"IX_ROBOT_PROT_DOOR_CLSD"	I 3111.3	BOOL	// F4-66.7 Werkstücklader Schutzzaun geschlossen
"MSST_Vorschub_OVR"	IB 3	BYTE	// Maschinensteuertafel Vorschub Override
"MSST_Eilgang_OVR"	IB 7	BYTE	// Maschinensteuertafel Eilgang Override
"IX_Direkttasten_links"	IB 8	BYTE	// HMI-PRO: OP12/OP15A Direkttasten links
"IX_Direkttasten_rechts"	IB 9	BYTE	// HMI-PRO: OP12/OP15A Direkttasten rechts
"IW_SPI_VIBRATION"	IW 100	WORD	// Analogeingang Vibrationssensor
"IW_FD_PT100"	IW 156	WORD	// Temperatursensor Pt100 Fraes-Drehtisch
"IW_MI_TURNT_TEMP"	IW 1000	WORD	// Temp.-Sensor PT100 Fraes-Drehtisch
"IW_MACH_BED_T_COMP"	IW 1090	WORD
"IW_SPI_TEMP_BEA_FRONT"	IW 1092	WORD
"IW_VMS_VIBRATION_SPINDLE"	IW 1094	WORD
"IW_SPI_LINE_PT100_1"	IW 1102	WORD	// Temperatursensor 1 Leitungsueberwachung Hauptantrieb
"IW_SPI_LINE_PT100_2"	IW 1104	WORD	// Temperatursensor 2 Leitungsueberwachung Hauptantrieb
"IW_SPI_PT100"	IW 1106	WORD	// Lager-Temperatursensor PT100 Hauptantrieb
"IW_HCD_PRE_MPL"	IW 1108	WORD	// Spannhydraulik Druckueberwachung Maschine
"IW_HCD_PRE_SST"	IW 1110	WORD	// Spannhydraulik Druckueberwachung Ruestplatz
"IW_SPI_TEMP_LAG_VORNE"	IW 1112	WORD	// Lager-Temperatursensor PT100 Hauptantrieb
"IW_SPI_TEMP_LAG_HINTEN"	IW 1122	WORD	// Lager-Temperatursensor PT100 Hauptantrieb
"IW_SPI_TEMP_MONITOR"	IW 2000	WORD	// Temperaturüberwachung Spindelstock (55/65H)
"IW_RESERVE_4_33"	IW 2002	WORD	// Dummy für Hardware 55H
"BT_ET200S_3_12"	IW 3106	WORD	// E5-03.5 Analogeingang Reserve
"BT_ET200S_4_5"	IW 3108	WORD	// Analogeingang Reserve
"m_null"	M 0.0	BOOL	// Status 0
"m_eins"	M 0.1	BOOL	// Status 1
"m_expertenbit"	M 0.2	BOOL	// Expertenbit für Fehleranzeige
"m_dummy"	M 0.3	BOOL	// Dummy
"m_vke_uebertrag_1"	M 0.4	BOOL	// VKE Übertrag 1
"m_neustart"	M 0.5	BOOL	// Neustart
"m_inbetrieb_logisch_1"	M 0.6	BOOL	// Inbetriebnahmemerker Logisch 1
"m_konstruktion"	M 0.7	BOOL	// Konstruktionsmerker Logisch 1
"m_takt_0,1sec."	M 1.0	BOOL	// Taktmerker System 100 ms
"m_takt_0,2sec."	M 1.1	BOOL	// Taktmerker System 200 ms
"m_takt_0,4sec."	M 1.2	BOOL	// Taktmerker System 400 ms
"m_takt_0,5sec."	M 1.3	BOOL	// Taktmerker System 500 ms
"m_takt_0,8sec."	M 1.4	BOOL	// Taktmerker System 800 ms
"m_takt_1sec."	M 1.5	BOOL	// Taktmerker System 1000 ms
"m_takt_1,6sec."	M 1.6	BOOL	// Taktmerker System 1600 ms
"m_takt_2sec."	M 1.7	BOOL	// Taktmerker System 2000 ms
"M_1_ter_OB1_Zyklus"	M 2.0	BOOL	// Erster Zyklus OrganisationsBaustein 1
"M_2_ter_OB1_Zyklus"	M 2.1	BOOL	// Zweiter Zyklus OrganisationsBaustein 1
"M_3_ter_OB1_Zyklus"	M 2.2	BOOL	// Dritter Zyklus OrganisationsBaustein 1
"M_4_ter_OB1_Zyklus"	M 2.3	BOOL	// Vierter Zyklus OrganisationsBaustein 1
"M_5_ter_OB1_Zyklus"	M 2.4	BOOL	// Fünfter Zyklus OrganisationsBaustein 1
"M_6_ter_OB1_Zyklus"	M 2.5	BOOL	// Sechster Zyklus OrganisationsBaustein 1
"M_7_ter_OB1_Zyklus"	M 2.6	BOOL	// Siebter Zyklus OrganisationsBaustein 1
"M_8_ter_OB1_Zyklen"	M 2.7	BOOL	// Achter Zyklus OrganisationsBaustein 1
"M_CHAN2_aktiv"	M 6.0	BOOL	// Kanal 2 aktiv
"m_6.1"	M 6.1	BOOL	// Reserve
"m_6.2"	M 6.2	BOOL	// Reserve
"m_6.3"	M 6.3	BOOL	// Reserve
"m_6.4"	M 6.4	BOOL	// Reserve
"m_6.5"	M 6.5	BOOL	// Reserve
"m_6.6"	M 6.6	BOOL	// Reserve
"M_Takt_10s"	M 6.7	BOOL	// Taktmerker 10 s
"M_Takt_01s"	M 7.0	BOOL	// Taktmerker 100 ms
"M_Takt_02s"	M 7.1	BOOL	// Taktmerker 200 ms
"M_Takt_04s"	M 7.2	BOOL	// Taktmerker 400 ms
"M_Takt_05s"	M 7.3	BOOL	// Taktmerker 500 ms
"M_Takt_08s"	M 7.4	BOOL	// Taktmerker 800 ms
"M_Takt_1s"	M 7.5	BOOL	// Taktmerker 1000 ms
"M_Takt_16s"	M 7.6	BOOL	// Taktmerker 1600 ms
"M_Takt_2s"	M 7.7	BOOL	// Taktmerker 2000 ms
"M_Takt_Speicher_01s"	M 8.0	BOOL	// Taktmerker Speicher 100 ms
"M_Takt_Speicher_02s"	M 8.1	BOOL	// Taktmerker Speicher 200 ms
"M_Takt_Speicher_04s"	M 8.2	BOOL	// Taktmerker Speicher 400 ms
"M_Takt_Speicher_05s"	M 8.3	BOOL	// Taktmerker Speicher 500 ms
"M_Takt_Speicher_08s"	M 8.4	BOOL	// Taktmerker Speicher 800 ms
"M_Takt_Speicher_1s"	M 8.5	BOOL	// TaktmerkerSpeicher 1000 ms
"M_Takt_Speicher_16s"	M 8.6	BOOL	// Taktmerker Speicher 1600 ms
"M_Takt_Speicher_2s"	M 8.7	BOOL	// Taktmerker Speicher 2000 ms
"M_1_ter_OB1_Zyklus_stat"	M 9.0	BOOL	// Erster Zyklus OrganisationsBaustein 1
"M_Ruecksetze_Fehler"	M 10.0	BOOL	// Globaler Reset fuer Fehler (Quitt Taste und Reset Taste)
"M_NC_Stop"	M 10.1	BOOL	// Globaler NC Stop
"M_Vorschub_Halt_Kanal"	M 10.2	BOOL	// Globaler Vorschub Halt
"M_Spindel_Halt_Kanal"	M 10.3	BOOL	// Globaler Spindel Halt
"M_Vorschub_Halt_Haupt"	M 10.4	BOOL	// Vorschub Halt Hauptachsen
"M_Reset_Taste"	M 10.5	BOOL	// Globaler Impuls Reset Taste
"M_Fehler_Quit_Taste"	M 10.6	BOOL	// Globaler Impuls Quittier Taste
"M_NC_Stop_Taste"	M 10.7	BOOL	// NC-Stop Taste in BA AUTO (nicht in Jog)
"M_NC_Start_Taste"	M 11.0	BOOL	// NC-Start Taste in BA AUTO (nicht in Jog)
"M_Spindel_Sperre_Auto"	M 11.1	BOOL	// Spindel-Sperre Taste in Automatik
"M_Vorschub_Sperre_Auto"	M 11.2	BOOL	// Vorschub-Sperre Taste in Automatik
"M_Eilgang_verriegeln"	M 11.3	BOOL	// Eilgangtaste verriegeln
"M_Vorschub_Halt_Asyn1"	M 11.4	BOOL	// Vorschub Halt Asynchroner Prozess 1 (701548-701631 -> Mag: Achse 7)
"M_Vorschub_Halt_Asyn2"	M 11.5	BOOL	// Vorschub Halt Asynchroner Prozess 2 (701632-701715 -> PW: Achse 8)
"M_Vorschub_Halt_Asyn3"	M 11.6	BOOL	// Vorschub Halt Asynchroner Prozess 3 (701716-701763 -> Pal.Speicher: Achse9/10)
"M_Vorschub_Halt_Asyn4"	M 11.7	BOOL	// Vorschub Halt Asynchroner Prozess 4 (701800-701847 ->  Mag: Achse 7)
"M_Handbetrieb"	M 12.0	BOOL	// Manual / Jog-betrieb steht an
"M_Satzfolge_aktiv"	M 12.1	BOOL	// Automatikbetrieb
"M_Einzelsatz"	M 12.2	BOOL	// Einzelsatz
"M_Simulation_Aktiv"	M 12.3	BOOL	// Simulation Aktiv
"M_Programm_Aktiv"	M 12.4	BOOL	// Programm Aktiv
"M_Hauptprogramm_Ende"	M 12.5	BOOL	// Hauptprogramm Ende
"M_HM_Hauptprogramm_Ende"	M 12.6	BOOL	// Hilfsmerker Hauptprogramm Ende
"M_Gewindeschneiden_aktiv"	M 12.7	BOOL	// Nahtstelle: Gewindeschneiden aktiv
"M_Hauptspindel_steht"	M 13.0	BOOL	// Hauptspindel steht
"M_Hauptachsen_stehen"	M 13.1	BOOL	// Hauptachsen stehen
"M_ShopMill_aktiv"	M 13.2	BOOL	// ShopMill Bedienoberflaeche aktiv
"M_FahrAnf_HauptAchs"	M 13.3	BOOL	// Fahranforderung Hauptachsen steht an
"M_G00_aktiv"	M 13.4	BOOL	// G0 Aktiv
"M_G02_G03_aktiv"	M 13.5	BOOL	// G02 oder G03 Aktiv
"M_G74_aktiv"	M 13.6	BOOL	// G74 Aktiv
"M_Automatik_Betrieb"	M 13.7	BOOL	// Automatikbetrieb steht an
"M_ShopMill_Manual"	M 14.0	BOOL	// ShopMill im Manual
"M_ShopMill_Positionieren"	M 14.1	BOOL	// ShopMill Positionieren
"MX_MsSt_Vorschub_0"	M 14.2	BOOL	// Anforderung MSST Vorschub Override auf 0
"MX_M0_1_Aktiv"	M 14.3	BOOL	// M0 oder M1 ist aktiv
"MX_Flanke_M01"	M 14.4	BOOL	// Flanke Positiv M0 M1
"MX_MDA"	M 14.5	BOOL	// MDA Aktiv
"MX_FN_Leistung_Steht_an"	M 14.6	BOOL	// Flanke Negativ Leistung
"MX_IMP_Leistung_0"	M 14.7	BOOL	// Flanke Negativ Leistung Steht an
"MX_SonderBA_Stop"	M 15.0	BOOL	// Stop Aktiv nach verlassen der Sonder BA's
"MX_PLC_Initialisiert"	M 15.1	BOOL	// PLC Initialisiert
"M_Programm_Aktiv_Kanal_1"	M 15.2	BOOL	// Programm aktiv im Kanal 1(Run/Wait/Stop/Interrupt)
"MX_Satzsuchlauf_gesp"	M 15.3	BOOL	// Satzsuchlauf aktiv gespeichert
"O_PW_TUER_ENTRIEGELN"	M 15.4	BOOL	// M-AUSGANG: Magnetverriegelung Ruestplatz Palettenwechsler verriegeln
"O_PW_Ventil_Abfrage"	M 15.5	BOOL	// M-AUSGANG: Ventil Luftstrom Palette
"M_G01_aktiv"	M 15.6	BOOL	// G1 Aktiv
"O_PW_Ventil_Tischspuel"	M 15.7	BOOL	// M-AUSGANG: IKZ-Pumpe ein für Tischspuelung
"I_MSST_PW_Freigabe"	M 16.0	BOOL	// M-EINGANG: Eingang Freigabe Palettenwechsler
"I_PW_MPL_belegt"	M 16.1	BOOL	// M-EINGANG: Palette in der Maschine vorhanden
"I_PW_Ruestpl_UeberG"	M 16.2	BOOL	// M-EINGANG: Palette Übergabeplatz Maschine
"I_PW_Hub_in_Mitte"	M 16.3	BOOL	// M-EINGANG: Palettenwechsler Hub Pos. Mitte
"I_PW_Tueren_verriegelt"	M 16.4	BOOL	// M-EINGANG: Fenster Ruestplatz PW verriegelt
"I_PW_Klemmung_Geklemmt"	M 16.5	BOOL	// M-EINGANG: Palettenklemmung geklemmt
"I_PW_Klemmung_Gelöst"	M 16.6	BOOL	// M-EINGANG: Palettenklemmung gelöst
"M_FLANKE_START_TASTE"	M 16.7	BOOL	// Flanke Positiv NC-Start Taste
"M_Flanke_M208"	M 17.0	BOOL	// TEMPERATURKOMPENSATION: M-Funktion 208 Flanke positiv
"M_Flanke_M209"	M 17.1	BOOL	// TEMPERATURKOMPENSATION: M-Funktion 209 Flanke positiv
"M_Umlaufzaehler=0"	M 17.3	BOOL	// TEMPERATURKOMPENSATION: Umlaufzähler HM
"M_Zyklus_Takt"	M 17.4	BOOL	// TEMPERATURKOMPENSATION: Zyklus Takt
"M_VSH_ASYN_DISABLE_START"	M 17.5	BOOL	// Ersten Start unterdrücken nach Vorschub Halt Asynchroner Prozess bei Fertigtteil
"m_17.6"	M 17.6	BOOL	// Reserve
"M_Fuehlerumschaltung"	M 17.7	BOOL	// TEMPERATURKOMPENSATION: Fühlerumschaltung
"M_Trend_Temp_auf"	M 18.0	BOOL	// TEMPERATURKOMPENSATION: Temperaturtrend aufwärts
"M_Trend_Temp_gleich"	M 18.1	BOOL	// TEMPERATURKOMPENSATION: Temperaturtrend gleichbleibend
"M_Trend_Temp_ab"	M 18.2	BOOL	// TEMPERATURKOMPENSATION: Temperaturtrend abwärts
"M_Fehler_Temp-Tabelle"	M 18.3	BOOL	// TEMPERATURKOMPENSATION: Fehler Temperaturtabelle
"M_FM_Timer_Verzoegerung"	M 18.4	BOOL	// TEMPERATURKOMPENSATION: Timer Verzögerung
"M_FP_Timer_Verzoegerung"	M 18.5	BOOL	// TEMPERATURKOMPENSATION: Timer Verzögerung Flanke positiv
"M_Temp-Daten_uebertragen"	M 18.6	BOOL	// TEMPERATURKOMPENSATION: Temperaturdaten übertragen
"M_MesswertInterv_0"	M 18.7	BOOL	// TEMPERATURKOMPENSATION: Messwert-Intervall  = 0
"M_Trend_Drehz_auf"	M 19.0	BOOL	// TEMPERATURKOMPENSATION: Drehzahltrend aufwärts
"M_Trend_Drehz_gleich"	M 19.1	BOOL	// TEMPERATURKOMPENSATION: Drehzahltrend gleichbleibend
"M_Trend_Drehz_ab"	M 19.2	BOOL	// TEMPERATURKOMPENSATION: Drehzahltrend abwärts
"M_Fehler_Drehz-Tabelle"	M 19.3	BOOL	// TEMPERATURKOMPENSATION: Fehler Drehzahltabelle
"M_Temp_Wert <"	M 19.4	BOOL	// TEMPERATURKOMPENSATION: Temperaturwert kleiner
"M_Temp_Wert ="	M 19.5	BOOL	// TEMPERATURKOMPENSATION: Temperaturwert gleich
"M_Temp_Wert >"	M 19.6	BOOL	// TEMPERATURKOMPENSATION: Temperaturwert größer
"HM_PI_Umlauf"	M 19.7	BOOL	// TEMPERATURKOMPENSATION:  PI Umlaufzähler = 0 Flanke positiv
"M_FP_Einrichtb"	M 20.0	BOOL	// Einrichtbetrieb Flanke positiv
"M_Imp_Einrichtberieb"	M 20.1	BOOL	// Einrichtbetrieb Impuls
"M_FP_BA3"	M 20.2	BOOL	// Betriebsart 3 Flanke positiv
"M_Imp_Betriebsart 3"	M 20.3	BOOL	// Betriebsart 3  Impuls
"M_FP_BA4+ZUSTT"	M 20.4	BOOL	// Betriebsart 4 Flanke positiv
"M_BA4_aktiv_schalten_"	M 20.5	BOOL	// Betriebsart 4  aktiv
"m_20.6"	M 20.6	BOOL	// Reserve
"m_20.7"	M 20.7	BOOL	// Reserve
"m_21.0"	M 21.0	BOOL	// Reserve
"m_21.1"	M 21.1	BOOL	// Reserve
"m_21.2"	M 21.2	BOOL	// Reserve
"m_21.3"	M 21.3	BOOL	// Reserve
"m_21.4"	M 21.4	BOOL	// Reserve
"m_21.5"	M 21.5	BOOL	// Reserve
"m_21.6"	M 21.6	BOOL	// Reserve
"m_21.7"	M 21.7	BOOL	// Reserve
"m_22.0"	M 22.0	BOOL	// Reserve
"M_Selbsth_AT_X-plus"	M 22.1	BOOL	// MSTT: Selbsthaltung für Achsenkreuztaste X-Plus
"M_Selbsth_AT_X-minus"	M 22.2	BOOL	// MSTT: Selbsthaltung für Achsenkreuztaste X-Minus
"m_22.3"	M 22.3	BOOL	// Reserve
"m_22.4"	M 22.4	BOOL	// Reserve
"m_22.5"	M 22.5	BOOL	// Reserve
"m_22.6"	M 22.6	BOOL	// Reserve
"m_22.7"	M 22.7	BOOL	// Reserve
"m_23.0"	M 23.0	BOOL	// Reserve
"m_23.1"	M 23.1	BOOL	// Reserve
"M_Selbsth_AT_Y-minus"	M 23.2	BOOL	// MSTT: Selbsthaltung für Achsenkreuztaste Y-Minus
"M_Selbsth_AT_Y-plus"	M 23.3	BOOL	// MSTT: Selbsthaltung für Achsenkreuztaste Y-Plus
"M_Selbsth_AT_Z-minus"	M 23.4	BOOL	// MSTT: Selbsthaltung für Achsenkreuztaste Z-Minus
"M_Selbsth_AT_Z-plus"	M 23.5	BOOL	// MSTT: Selbsthaltung für Achsenkreuztaste Z-Plus
"M_Selbsth_AT_4-minus"	M 23.6	BOOL	// MSTT: Selbsthaltung für Achsenkreuztaste 4-Minus
"M_Selbsth_AT_4-plus"	M 23.7	BOOL	// MSTT: Selbsthaltung für Achsenkreuztaste 4-Plus
"M_Selbsth_AT_5-minus"	M 24.0	BOOL	// MSTT: Selbsthaltung für Achsenkreuztaste 5-Minus
"M_Selbsth_AT_5-plus"	M 24.1	BOOL	// MSTT: Selbsthaltung für Achsenkreuztaste 5-Plus
"M_Selbsth_AT_6-minus"	M 24.2	BOOL	// MSTT: Selbsthaltung für Achsenkreuztaste 6-Minus
"M_Selbsth_AT_6-plus"	M 24.3	BOOL	// MSTT: Selbsthaltung für Achsenkreuztaste 6-Plus
"M_Selbsth_AT_10-minus"	M 24.4	BOOL	// MSTT: Selbsthaltung für Achsenkreuztaste 10-Minus
"M_Selbsth_AT_10-plus"	M 24.5	BOOL	// MSTT: Selbsthaltung für Achsenkreuztaste 10-Plus
"O_SP_RPL_MPL_BLASLUFT"	M 24.6	BOOL	// M-AUSGANG: Ventil Blasluft Medienkupplung
"M_FP_mxplus"	M 24.7	BOOL	// Flanke Positiv Achsenkreuztaste X-Plus
"M_FP_mxminus"	M 25.0	BOOL	// Flanke Positiv Achsenkreuztaste X-Minus
"M_FP_myplus"	M 25.1	BOOL	// Flanke Positiv Achsenkreuztaste Y-Plus
"M_FP_myminus"	M 25.2	BOOL	// Flanke Positiv Achsenkreuztaste Y-Minus
"M_FP_mzplus"	M 25.3	BOOL	// Flanke Positiv Achsenkreuztaste Z-Plus
"M_FP_mzminus"	M 25.4	BOOL	// Flanke Positiv Achsenkreuztaste Z-Minus
"M_FP_m6plus"	M 25.5	BOOL	// Flanke Positiv Achsenkreuztaste 6-Plus
"MX_BHG_Lampentest"	M 25.6	BOOL	// BHG MPI: Lampentest
"M_FP_m6minus"	M 25.7	BOOL	// Flanke Positiv Achsenkreuztaste 6-Minus
"M_FP_m4plus"	M 26.0	BOOL	// Flanke Positiv Achsenkreuztaste 4-Plus
"M_FP_m4minus"	M 26.1	BOOL	// Flanke Positiv Achsenkreuztaste 4-Minus
"M_FP_m5plus"	M 26.2	BOOL	// Flanke Positiv Achsenkreuztaste 5-Plus
"M_FP_m5minus"	M 26.3	BOOL	// Flanke Positiv Achsenkreuztaste 5-Minus
"M_FP_m10plus"	M 26.4	BOOL	// Flanke Positiv Achsenkreuztaste 10-Plus
"M_FP_m10minus"	M 26.5	BOOL	// Flanke Positiv Achsenkreuztaste 10-Minus
"m_26.6"	M 26.6	BOOL	// Reserve
"m_26.7"	M 26.7	BOOL	// Reserve
"m_27.0"	M 27.0	BOOL	// Reserve
"m_27.1"	M 27.1	BOOL	// Reserve
"m_27.2"	M 27.2	BOOL	// Reserve
"m_27.3"	M 27.3	BOOL	// Reserve
"m_27.4"	M 27.4	BOOL	// Reserve
"m_27.5"	M 27.5	BOOL	// Reserve
"m_27.6"	M 27.6	BOOL	// Reserve
"m_27.7"	M 27.7	BOOL	// Reserve
"m_28.0"	M 28.0	BOOL	// Reserve
"m_28.1"	M 28.1	BOOL	// Reserve
"m_28.2"	M 28.2	BOOL	// Reserve
"M_NCStop_anfordern"	M 28.3	BOOL	// NC-Stop anfordern
"m_28.4"	M 28.4	BOOL	// Reserve
"m_28.5"	M 28.5	BOOL	// Reserve
"m_28.6"	M 28.6	BOOL	// Reserve
"m_28.7"	M 28.7	BOOL	// Reserve
"MX_FP_WZW_Aktiv"	M 36.0	BOOL	// Flanke Positiv WZW aktiv
"MX_WZW_RPC_START"	M 36.1	BOOL	// PI Start Werkzeug auswechseln an RPC
"mx_Pal_status_okay"	M 36.3	BOOL	// Meldung Status Palette von RPC okay(Staus <> 0)
"M_M3oderM4"	M 45.3	BOOL	// M3 oder M4 aktiv
"M_NCStop_aktiv"	M 51.0	BOOL	// NC-Stop von MSST ist aktiv
"HM_PI_Taste_X_Anwahl"	M 51.3	BOOL	// BHG-MPI: Taste X-Anwahl Flanke positiv
"HM_PI_Taste_C_Anwahl"	M 51.4	BOOL	// BHG-MPI: Taste C-Anwahl Flanke positiv
"HM_PI_BHG_Anf_JOG"	M 51.5	BOOL	// BHG-MPI: Anforderung JOG Flanke positiv
"I_WW_1_ZYL_GST"	M 52.5	BOOL	// M-EINGANG: WW Pneumatikzylinder 1 Grundstellung
"m_55.0"	M 55.0	BOOL	// WZB: Reserve
"MX_WZB_Toleranz"	M 55.1	BOOL	// WZB: Toleranz zwischen 1. u. .2. Messung > zu gross
"MX_WZB_2MW_gr_1MW"	M 55.2	BOOL	// WZB: 2.Messwert > 1. Messwert
"MX_WZB_NeuWahl"	M 55.3	BOOL	// WZB: Neuwahl eines vorbereiteten WZ
"MX_T_WechselRdy"	M 55.4	BOOL	// WZB: T wurde eingewechselt
"MX_WZB_Ov_0"	M 55.5	BOOL	// WZB: Override auf 0
"MX_WZB_Anf_Lesen"	M 55.6	BOOL	// WZB: Anforderung Lesen
"MX_WZB_Fertig_Lesen"	M 55.7	BOOL	// WZB: Fertigmeldung Lesen
"M_WZW_Hub_Magazin_2"	M 56.5	BOOL	// Längsachse auf Position Magazin 2
"M_WZW_Hub_Magazin"	M 58.0	BOOL	// WZW: Querhubachse Hub am Magazin
"M_WZW_Hub_GrdSt"	M 58.1	BOOL	// WZW: Querhubachse Hub in Grundstellung
"I_KA2_N_STOERMELDUNG1"	M 58.2	BOOL	// M-EINGANG: Kuehlaggregat 2 Störmeldung Prioritaet 1
"M_Umsp_Spdl-Mag"	M 58.3	BOOL	// WZV: Umspeichern von Spindel in Magazin
"M_IMP_INIT_Fertig"	M 58.4	BOOL	// MESS: Impuls Init fertig
"I_KA2_N_STOERMELDUNG2"	M 58.5	BOOL	// M-EINGANG: Kuehlaggregat 2 Störmeldung Prioritaet 2
"I_KA2_N_WARNMELDUNG"	M 58.6	BOOL	// M-EINGANG: Kuehlaggregat 2 Warnmeldung
"M_Umsp_Gr1-Spdl"	M 58.7	BOOL	// WZV: Umspeichern von Greifer1 in Spindel
"M_Umsp_Spdl_Gr2"	M 59.0	BOOL	// WZV: Umspeichern von Spindel in Greifer 2
"O_WW_1_ZYL_SPI"	M 59.2	BOOL	// M-AUSGANG: Werkzeugmagazin Zylinder1 Richtung Spindel / Richtung Magazin
"O_WW_1_ZYL_GST"	M 59.3	BOOL	// M-AUSGANG: Werkzeugmagazin Zylinder1 Richtung Grundstellung
"I_WW_1_ZYL_WZM"	M 59.4	BOOL	// M-EINGANG: WW Pneumatikzylinder 1 Werkzeugmagazin
"M_WZW_Sperre_ZB"	M 59.5	BOOL	// WZW: Sperre Wechsel Betriebsart
"M_WZW_Hub_Magazin_1"	M 59.6	BOOL	// Längsachse auf Position Magazin 1
"MX_WZB_G0_Sperre"	M 59.7	BOOL	// WZB: Werkzeugbruch G0 Sperre
"Mx_Imp_H47"	M 67.0	BOOL	// H-Funktion 47 Flanke positiv
"Mx_H47_angefordert"	M 67.7	BOOL	// H-Funktion 47 angefordert ->  Potis mittels H-Funktion (Wert1-3) auf 100%
"M_Kabine_verriegeln"	M 70.0	BOOL	// Kabinentüre verriegeln
"I_AL_HYD_FUELLMAX_TEMP"	M 70.1	BOOL	// M-EINGANG: Fuellstand Hydraulik Max. / Hydraulik Temperaturueberwachung
"M_Freigabe_ZD_WZW"	M 70.2	BOOL	// WZW: Achsen in sicherer Position
"Mx_PW_Werkstückspülung"	M 70.4	BOOL	// PW: Werkstückspülung ein
"Mx_Vert_Bremse_auf"	M 82.0	BOOL	// AX: Vertikale Achse Bremse öffnen
"Mx_horz_BRemse_Auf"	M 82.1	BOOL	// AX: Horizontale Bremse (Z-Achse öffnen)
"M_NC_Konus_ausblasen"	M 82.2	BOOL	// $A_OUT[33] Befehl von NC Konus ausblasen
"Mx_XAchse_Bremse_Auf"	M 82.3	BOOL	// AX: X-Achse Bremse öffnen
"M_PS_HUB_AX_Bremse_auf"	M 82.4	BOOL	// AX: Palettenspeicher Hub-Achse Bremse öffnen
"I_WZ_MIN_SCH_DRUCK_OK"	M 83.0	BOOL	// M-EINGANG: Minimalmengenschmierung Druck ok
"M_MWZW_Tuer_Auf"	M 83.1	BOOL	// MAN WZW: Entriegeln Tuer
"M_Umsp_Gr2-Mag"	M 83.2	BOOL	// WZV: Umspeichern WZ in Magazin
"O_WZ_MIN_SCH_MV2"	M 83.3	BOOL	// M-AUSGANG: Minimalmengen Schmierung Ventil 2 Ein
"I_KM_DRUCK0_M7_EIN"	M 83.4	BOOL	// M-EINGANG: Kuehlmittel Freigabe Maschine Druckstufe 0
"I_PW_UPL_PAL_VORH"	M 83.5	BOOL	// M-EINGANG: Palette auf PW-Übergabeplatz vorhanden (bei Palettenspeicher)
"MX_I_Palette_auf_UG"	M 83.6	BOOL	// PW: Ruestplatz Wechselposition + Palette auf PW-Übergabeplatz vorhanden
"M_PF_ZImp"	M 84.0	BOOL	// GT MAG: Positive Flanke Zaehlimpuls
"M_NF_ZImp"	M 84.1	BOOL	// GT MAG: Negative Flanke ZaehlImpuls
"M_WZ_Spanner_Zu_Ohne_WZ"	M 84.2	BOOL	// WZW: WZ-Spanner geschlossen ohne WZ
"M_WZW_Prozess_Aktiv"	M 84.3	BOOL	// WZW: Aktiver Prozess
"M_Umsp_Mag-Gr1"	M 84.4	BOOL	// WZV: Umspeichern Magazin-Greifer 1
"M_WZW_Fehler_Grdst"	M 84.5	BOOL	// WZW: Fehler Grundstellung
"M_Umsp_Mag-Gr2"	M 84.6	BOOL	// WZV: Umspeichern Magazin-Greifer 2
"MX_Lesen_MagPos"	M 84.7	BOOL	// MAG: Lesen Magazinposition - > TDS BALLUFF
"MX_RDY_Lesen_MagPos"	M 85.0	BOOL	// MAG: Ready Lesen Magazinposition -> TDS BALLUFF
"MX_TDS_Aktiv"	M 85.1	BOOL	// TDS: Aktiv
"MX_TDS_MagSperre"	M 85.2	BOOL	// TDS: Magazin Sperre
"MX_BeEntladen_Aktiv"	M 85.3	BOOL	// WZV: Be.-Entladen aktiv
"MX_TMAG_Anforderung"	M 85.4	BOOL	// WZV: Anforderung T (Magazin)
"MX_TMAG_Fertig"	M 85.5	BOOL	// WZV: Fertig T (Magazin)
"MX_TMMAG_Anforderung"	M 85.6	BOOL	// WZV: Anforderung TM (Magazin)
"MX_TMMAG_Fertig"	M 85.7	BOOL	// WZV: Fertig TM (Magazin)
"M_Mag_Inposition"	M 99.0	BOOL	// GT MAG: Magazin in Position
"M_Mag_Kalibriert"	M 99.1	BOOL	// GT MAG: Magazin Kalibriert
"M_GT_MAG_Trigg1"	M 99.2	BOOL	// GT MAG: Trigger 1 (FC_GT_MAG_STAT)
"M_GT_MAG_Trigg2"	M 99.3	BOOL	// GT MAG: Trigger 2 (FC_GT_MAG_ABL)
"M_GT_MAG_Trigg3"	M 99.4	BOOL	// GT MAG: Trigger 3 (FC_GT_MAG_ABL)
"M_MAG_Schalter_Gueltig"	M 99.6	BOOL	// GT MAG: Schalter gueltig
"M_GT_MAG_Trigg4"	M 99.7	BOOL	// GT MAG: Trigger 4 (FC_MAG_HAUPT_ZH)
"MX_Mag_Trigg2"	M 104.0	BOOL	// MAG: Trigger 2  (FC_MAG_HAUPT_ZH)
"MX_Mag_Trigg3"	M 104.1	BOOL	// MAG: Trigger 3  (FC_MAG_HAUPT_ZH)
"O_WZ_MIN_SCH_Ums_M8"	M 104.2	BOOL	// M-AUSGANG: Umschaltung Ventil Schmiersystem Kuehlmittel 1
"MX_Req_Reinigen_Abl"	M 104.3	BOOL	// WZW: Anforderung Reinigen und Ablegen
"MX_Rdy_Reinigen_Abl"	M 104.4	BOOL	// WZW: Rückmeldung Reinigen und Ablegen
"MX_Mag_Pos_Gueltig"	M 104.5	BOOL	// MAG: Magazinposition gueltig
"MX_Anf_Reinin_InWZW"	M 104.6	BOOL	// MAG: Anforderung Reinigen bei WZW
"O_WZ_MIN_SCH_Ums_M7"	M 104.7	BOOL	// M-AUSGANG: Umschaltung Ventil Schmiersystem innere Kuehlmittelzufuhr
"I_MAS_SPANNDUCK_OK"	M 105.0	BOOL	// M-EINGANG: Druckschalter Spannvorrichtung gespannt
"MX_M47_Aktiv"	M 105.1	BOOL	// WZW: M47 (HSK Kegelreinigen) ist aktiv
"I_PW_RPL_SPANNDRUCK_OK"	M 105.2	BOOL	// M-EINGANG: Spanndruck Ruestplatz vorhanden
"M_Start_Kratzf"	M 105.3	BOOL	// KM: Start Kratzförderer bei Maschine Ein alle 30 Minuten
"MX_WZW_Mag_Verrieg"	M 105.4	BOOL	// WZW: Magazin Verriegelung
"m_wwgf_RqMagPos"	M 105.5	BOOL	// Wzw Grundstlg.fahren:Magazin Pos. anfahren
"M_WZW_FRG_AN_MAG"	M 105.6	BOOL	// WZW:  Werkzeugwechsler in Grundstellung (Freigabe zum Fahren an Magazin)
"M_VORSCH_FREIG"	M 107.0	BOOL	// BA: Vorschubfreigaben ein
"M_Temp_VHH"	M 107.1	BOOL	// FC_CHAN1: Vorschub Halt
"M_FP_HR_bereit"	M 107.2	BOOL	// BHG: Handrad bereit in Stellung 5 Flanke positiv
"HM_NI_Taste_MAG_Zweihand"	M 107.3	BOOL	// MAG: Taste Magazin Zweihand-Bedienung Flanke negativ
"HM_PI_allg_Ueberw"	M 110.0	BOOL	// WZ-Ueberlast Monitoring Mode Flanke positiv
"m_wwgf_wwRset"	M 110.1	BOOL	// Wzw Grundstlg.fahren:Wzw-Reset
"m_wwgf_Gr1Spi"	M 110.2	BOOL	// Wzw Grundstlg.fahren:Grf.1 zur Spi.fahren
"m_wwgf_Gr1Mag"	M 110.3	BOOL	// Wzw Grundstlg.fahren:Grf.1 zum Mag.fahren
"m_wwgf_SpiSpa"	M 110.4	BOOL	// Wzw Grundstlg.fahren:Spindel spannen
"m_wwgf_Gr2entr"	M 110.5	BOOL	// Wzw Grundstlg.fahren:Grf.2 entriegeln
"m_wwgf_BruchGf"	M 110.6	BOOL	// Wzw Grundstlg.fahren:Bruchktrl.zurück
"m_wwgf_ReinGf"	M 110.7	BOOL	// Wzw Grundstlg.fahren:WzReinigung zurück
"M_FP_U_NotBetr"	M 111.0	BOOL	// AX: U-Achse aktivieren über Taste Flanke positiv
"m_ReqNckRes"	M 111.1	BOOL	// Anforderung NCK-Reset
"m_wwgf_WzHubGf"	M 111.2	BOOL	// Wzw Grundstlg.fahren:WzHub zurück
"m_wwgf_WzwvGf"	M 111.3	BOOL	// Wzw Grundstlg.fahren:Wz-Verriegelung am Übergabeplatz zurück
"m_wwgf_XArbRaum"	M 111.4	BOOL	// Wzw Grundstlg.fahren:X-Achse zum Arbeitsraum fahren
"m_wwgf_Tzu"	M 111.5	BOOL	// Wzw Grundstlg.fahren:WzwTür schliessen
"m_wwgf_SpiZNcLoe"	M 111.6	BOOL	// Wzw Grundstlg.fahren:Spi.in den zuletzt von Nc geford.Zust.stellen:Lösen
"m_wwgf_SpiZNcSpa"	M 111.7	BOOL	// Wzw Grundstlg.fahren:Spi.in den zuletzt von Nc geford.Zust.stellen:Spannen
"M_positiveFlankeE4.5"	M 112.0	BOOL	// Taste Achsanwahl Umschaltung Flanke positiv
"M_posFlankeE4.5_1Zyklus"	M 112.1	BOOL	// Taste Achsanwahl Umschaltung Impuls
"M_5o6Achse"	M 112.2	BOOL	// BHG: Spindel(true) oder 5-te Achse(false) angewaehlt
"m_wwgf_RGrRqVp"	M 112.3	BOOL	// WZW Grundstlg.fahren: Regalgreifer Vorposition anfahren
"M_FN_Kabine_ZU"	M 112.4	BOOL	// Kabinentüre geschlossen Flanke negativ
"m_wwgf_RGrRqWp"	M 112.5	BOOL	// WZW Grundstlg.fahren: Regalgreifer Wechselposition anfahren
"m_wwgf_RegGf"	M 112.6	BOOL	// WZW Grundstlg.fahren: Regalgreifer zur Gasse bzw. Regal Init/Gst.fahren
"m_wwgf_SkStrt"	M 112.7	BOOL	// WZW Grundstlg.fahren: Schrittkette Start
"I_AL_NEBELABSCH_EIN"	M 113.0	BOOL	// M-EINGANG: Nebel- u.Rauchabscheider Ein
"HM_PI_Bew_68_Minus"	M 113.1	BOOL	// WZW: HMI-Beweg.Minus: X-Achse zum Arbeitsraum Flanke positiv
"HM_PI_X_AX_auf_WFKpos"	M 113.2	BOOL	// WZW: HMI-Beweg.Plus: X-Achse zur WFK-Wechselposition Flanke positiv
"HM_PI_Bew_69_Plus"	M 113.3	BOOL	// WZW: HMI-Beweg.Plus:Vertikalachse zur WFK-Auswechselposition Flanke positiv
"I_AL_NEG_NEBELAB_FREI"	M 113.4	BOOL	// M-EINGANG: Nebel- u.Rauchabscheider Ein Schalter
"I_AL_NEG_MSS_NEBELABSCH"	M 113.5	BOOL	// M-EINGANG: Motorschutzschalter Nebel- u.Rauchabscheider
"O_AL_NEBELABSCH_EIN"	M 113.6	BOOL	// M-AUSGANG: Nebel- u.Rauchabscheider 'Ein'
"M_FP_Quit_Bereitst"	M 113.7	BOOL	// WZV: Quittierung Bereitstellen fertig Flanke positiv
"HM_PI_Bew_70_Plus"	M 114.0	BOOL	// WZW: HMI-Beweg.Plus:Spindel zur Wechselposition Flanke positiv
"Mx_RFG_FD_Tisch"	M 114.1	BOOL	// AX: Reglerfreigabe FD Tisch (Achse 4 bzw. C-Achse)
"I_KA_NEG_Wasserstand"	M 114.2	BOOL	// M-EINGANG: Kuehlaggregat Stoerung Fuellstand
"I_KA_NEG_Stroemungsw"	M 114.3	BOOL	// M-EINGANG: Kuehlaggregat Stoerung Durchflusswaechter
"I_KA_NEG_Temp"	M 114.4	BOOL	// M-EINGANG: Kühlaggregat Stoerung Temperaturregler
"I_KA_NEG_ND_Fehler"	M 114.5	BOOL	// M-EINGANG: Kuehlaggregat Stoerung Niederdruckbegrenzung
"I_KA_NEG_HD_Fehler"	M 114.6	BOOL	// M-EINGANG: Kuehlaggregat Stoerung Hochdruckbegrenzung
"HM_PI_Bew_14_Minus"	M 114.7	BOOL	// HM PI Bwegung  14 Minus
"HM_PI_X_WechPos"	M 115.0	BOOL	// HM PI X auf WW_pos
"HM_PI_Bew_14_Plus"	M 115.1	BOOL	// HM PI Bewegung 14 Plus
"HM_PI_X_WartePos"	M 115.2	BOOL	// HM PI X auf Warteposition
"HM_PI_Bew_15_Minus"	M 115.3	BOOL	// HM PI Bewegung 15 Minus
"HM_PI_Bew_15_Minus_Tel"	M 115.4	BOOL	// HM PI Bewegung 15 Minus bei FC_WW_Teller
"HM_PI_Bew_16_Plus"	M 115.5	BOOL	// HM PI Bewegung 16 Plus
"HM_PI_Bew_16_plus_Tel"	M 115.6	BOOL	// HM PI Bewegung 16 Plus FC_WW_Teller
"m_vwgf_MagTUnlock"	M 120.0	BOOL	// Wz am autom.Magazinwechselplatz entriegeln
"m_vwgf_GrEin"	M 120.1	BOOL	// Wzw Grundstlg.fahren:Greifer einfahren
"m_vwgf_GrAus"	M 120.2	BOOL	// Wzw Grundstlg.fahren:Greifer ausfahren
"m_vwgf_stpAsup1"	M 121.0	BOOL	// Wzw Grundstlg.fahren: Flanke Halt ASUP_MACHINE Nr.1
"m_vwgf_SpiLoe"	M 121.1	BOOL	// Wzw Grundstlg.fahren:Spindel lösen
"m_vwgf_TpuRTool"	M 121.2	BOOL	// Wzw Grundstlg.fahren:Tpu Stlg.release Tool anfahren
"m_vwgf_TpuGTool"	M 121.3	BOOL	// Wzw Grundstlg.fahren:Tpu Stlg.get Tool anfahren
"m_vwgf_TpuMagP"	M 121.4	BOOL	// Wzw Grundstlg.fahren:Tpu Stlg.Magazingpos.anfahren
"m_vwgf_TpuTrP"	M 121.5	BOOL	// Wzw Grundstlg.fahren:Tpu Stlg.Transferpos (Übergabe-/nahmepos.zu Grf) anfahren
"m_vwgf_MagTLock"	M 121.6	BOOL	// Wz am autom.Magazinwechselplatz verriegeln
"m_vwgf_UpGrTpu"	M 121.7	BOOL	// Wzw Grundstlg.fahren:Umspeichern Grf.[bei Tpu] nach Tpu
"Mx_Rückmelde_M190_Fkt"	M 124.0	BOOL
"M_SPI_RESTW_LOESCH_M30"	M 124.1	BOOL	// Spindel Restweg löschen bei M30 (Solutionline)
"MX_FP_PW_HUB_VOR_MITTE"	M 124.2	BOOL	// PW: Hub vor Mitte Flanke positiv
"MX_FN_PW_HUB_VOR_MITTE"	M 124.3	BOOL	// PW: Hub vor Mitte Flanke negativ
"MX_FP_PW_HUB_VOR_UNTEN"	M 124.4	BOOL	// PW: Hub vor Unten Flanke positiv
"MX_FN_PW_HUB_VOR_UNTEN"	M 124.5	BOOL	// PW: Hub vor Mitte Flanke negativ
"MX_PW_HUB_VOR_UNTEN_HEBE"	M 124.6	BOOL	// PW: Hub vor Unten heben Impuls
"MX_PW_HUB_VOR_UNTEN_SENK"	M 124.7	BOOL	// PW: Hub vor Unten senken Impuls
"MX_Blum_C_sperren"	M 126.0	BOOL	// LA: Sperre C-Achse wenn Laser ausgefahren
"I_KM_NEG_MSS_KSA"	M 126.1	BOOL	// M-EINGANG: Stoermeldung Kuehlmittelanlage Vorschub Halt
"I_KM_TPF_MOTOR_EIN"	M 126.2	BOOL	// M-EINGANG: Motor Papierbandfilter Ein
"M_Tool_Req"	M 126.3	BOOL	// SPINDEL: Werkzeugnummer hat sich geaendert
"M_Grf2_verz_verriegelt"	M 126.4	BOOL	// WZV: Greifer 2 verriegelt verzögert
"M_PS_Achsen_stehen"	M 126.6	BOOL	// Achsen im Bereich Palettenspeicher stehen
"I_RefImp_WZ_Mag"	M 126.7	BOOL	// M-EINGANG: Refernzpunkt Impuls Magazin
"I_KM_TPF_PAPIER_ENDE"	M 127.0	BOOL	// M-EINGANG: Filterband Ende
"I_KM_TPF_PAPIER_WARN"	M 127.1	BOOL	// M-EINGANG: Warnung Filterband Ende
"O_KM_TPF_MOTOR_EIN"	M 127.2	BOOL	// M-AUSGANG: Motor Ein Papierbandfilter
"M_Zusatzachsen_stehen"	M 127.3	BOOL	// Zusatzachsen im Bereich Maschine stehen
"Mx_Vorschub_HALT_SOKO"	M 127.4	BOOL	// SONDERKONSTRUKTION: Vorschub Halt von SOKO
"I_D_KM_TPF_MOTOR_EIN"	M 127.5	BOOL	// M-EINGANG: Stoerung Papierbandfilter
"I_SF_NEG_MSS"	M 127.6	BOOL	// M-EINGANG: Motorschutzschalter Spaenefoerderer Kratzerfoerderer
"I_KM_NEG_KSA_MELDUNG"	M 127.7	BOOL	// M-EINGANG: keine Stoerung Kuehlmittelanlage
"I_A_KM_TPF_PAPIER_ENDE"	M 128.0	BOOL	// M-EINGANG: Antivalente Ueberwachung Filterband Ende
"I_A_KM_TPF_PAPIER_WARN"	M 128.1	BOOL	// M-EINGANG: Antivalente Ueberwachung Papiermangel
"M_Start_Pos_M1"	M 129.0	BOOL	// WZV Teller: Start Positionieren Magazin 1
"M_Start_Pos_M2"	M 129.1	BOOL	// WZV Teller: Start Positionieren Magazin 2
"I_PW_Freigabe"	M 129.2	BOOL	// M-EINGANG: Freigabe Drehpalettenwechsler
"M_Anf_ART_oeffnen"	M 129.3	BOOL	// WZW Spanner: Anforderung Arbeitsraumtüre öffnen
"M_Sp_OVR_0"	M 129.4	BOOL	// WZW Spanner: Spindeloverride 0 nach Werkzeug spannen
"MX_Override100"	M 129.5	BOOL	// M-Funktion 147 -> Override auf 100% stellen (Reset mit M148)
"MA_Ready_Schmier"	M 136.2	BOOL	// MA: Ready Schmierzyklus
"MA_Req_Schmier"	M 136.3	BOOL	// MA: Request Schmierzyklus
"M_MA_FP_Maschine_Ein"	M 136.4	BOOL	// MA: Flanke Positiv Maschine Ein
"M_MA_FN_Maschine_Ein"	M 136.5	BOOL	// MA: Flanke Negativ Maschine Ein
"M_MA_Maschine_Ein"	M 136.6	BOOL	// MA: Maschine Ein
"M_MA_Hydr_Fehler"	M 136.7	BOOL	// MA: Fehler Hydraulik
"M_FP_ext_Taste_Tuer_verr"	M 137.0	BOOL	// HM positive Flanke externe Taste Arbeitsraumtuer verriegeln
"M_Kab_Tuer_Entr_MFKTgesp"	M 137.1	BOOL	// Kabinentüre entriegeln durch M-Funktion gespeichert
"M_Kab_Tuer_Entr"	M 137.2	BOOL	// MA: Kabinentür automatisch entriegeln
"M_Tuer_Trigg1"	M 137.3	BOOL	// MA: Kabinentür zu Flanke positiv
"M_Spritz_Tuer_Zu"	M 137.4	BOOL	// MA: Kabinentür geschlossen und verriegelt
"M_3Te_Betriebsart"	M 137.5	BOOL	// MA: 3. Betriebsart aktiv
"M_4Te_Betriebsart"	M 137.6	BOOL	// MA: 4. Betriebsart aktiv
"M_Einrichtbetrieb"	M 137.7	BOOL	// MA: Einrichtbetrieb aktiv
"M_Leistung_Steht_an"	M 138.0	BOOL	// MA: Leistung steht an
"M_FMN_Sonder_BA"	M 138.1	BOOL	// MA: Sonderbetriebsart aktiv Flanke negativ
"M_FP_Taste_Tuerver"	M 138.2	BOOL	// MA: Kabinentür entriegeln Flanke positiv
"M_FN_Leistung_Einricht"	M 138.3	BOOL	// MA: Einrichtbetrieb + Leistung Flanke negativ
"M_M5_Einrichtbetrieb"	M 138.4	BOOL	// MA: M5 (Spindel Halt) Anforderung von Einrichtbetrieb
"M_Taste_Tuerverieg"	M 138.5	BOOL	// MA: Taste Tuerverriegelung
"M_FM_3Te_Betriebsart"	M 138.6	BOOL	// MA: 3.Betriebsart aktiv Flanke positiv
"M_IMP_3Te_Betriebsart"	M 138.7	BOOL	// MA: 3.Betriebsart aktiv Impuls
"M_FM_4Te_Betriebsart"	M 139.0	BOOL	// MA: 4.Betriebsart aktiv Flanke positiv
"M_IMP_4Te_Betriebsart"	M 139.1	BOOL	// MA: 4.Betriebsart aktiv Impuls
"M_FM_Einrichtbetrieb"	M 139.2	BOOL	// MA: Betriebsart Einrichten aktiv Flanke positiv
"M_IMP_Einrichtbetrieb"	M 139.3	BOOL	// MA: Betriebsart Einrichten aktiv Impuls
"M_FMN_SonderBetriebsart"	M 139.4	BOOL	// MA: Keine Sonderbetriebsart aktiv Flanke positiv
"M_IMN_SonderBetriebsart"	M 139.5	BOOL	// MA: Keine Sonderbetriebsart aktiv Impuls
"M_FM_Leistung_steht_an"	M 139.6	BOOL	// MA: Leistung steht an Flanke positiv
"M_IMP_Leistung_steht_an"	M 139.7	BOOL	// MA: Leistung steht an Impuls
"O_AL_XACHS_Bremse_auf"	M 140.1	BOOL	// M-AUSGANG: Ansteuerung Motorbremse X-Achse
"O_WW_GRF_Drehen_fast"	M 140.2	BOOL	// M-AUSGANG: Werkstueckgreifer drehen schnell
"O_AL_YACHS_Bremse_auf"	M 140.3	BOOL	// M-AUSGANG: Ansteuerung Motorbremse Y-Achse
"O_WW_GRF_Drehen_slow"	M 140.4	BOOL	// M-AUSGANG: Werkstueckgreifer drehen langsam
"O_AL_ZACHS_Bremse_auf"	M 140.5	BOOL	// M-AUSGANG: Ansteuerung Motorbremse Z-Achse
"O_WW_1GRF_MAG"	M 140.6	BOOL	// M-AUSGANG: Werkzeuggreifer drehen Richtung Werkzeugmagazin
"O_AL_4ACHS_Bremse_auf"	M 140.7	BOOL	// M-AUSGANG: Ansteuerung Motorbremse 4-Achse
"O_AL_5ACHS_Bremse_auf"	M 141.1	BOOL	// M-AUSGANG: Ansteuerung Motorbremse 5-Achse
"M_Gewindeschneid_aktiv"	M 141.2	BOOL	// SPINDEL: Übergabe-Merker Gewindeschneiden Aktiv
"O_PW_ACHS_Bremse_auf"	M 141.5	BOOL	// M-AUSGANG: Achse 8 (PW)  Bremse lüften
"O_Bremse_oeffnen_Ax_7"	M 141.6	BOOL	// M-AUSGANG: Achse 7 Bremse lüften
"M_WZW_GRF_Beweg"	M 141.7	BOOL	// WZW: Greifer Bewegung
"M_Anf_Eilgang"	M 142.0	BOOL	// MSST: Anforderung Taste Eilgang
"M_Verfahrtaste gedrueckt"	M 142.1	BOOL	// MSST: Eine Achsverfahrtaste gedrueckt
"MX_1Zykl_M180"	M 142.2	BOOL	// MZU: 1 Zyklus verzögert M-Funktion 180
"MX_1Zykl_M181"	M 142.3	BOOL	// MZU: 1 Zyklus verzögert M-Funktion 181
"MX_1Zykl_M182"	M 142.4	BOOL	// MZU: 1 Zyklus verzögert M-Funktion 182
"MX_1Zykl_M183"	M 142.5	BOOL	// MZU: 1 Zyklus verzögert M-Funktion 183
"MX_1Zykl_M184"	M 142.6	BOOL	// MZU: 1 Zyklus verzögert M-Funktion 184
"MX_1Zykl_M185"	M 142.7	BOOL	// MZU: 1 Zyklus verzögert M-Funktion 185
"MX_1Zykl_M186"	M 143.0	BOOL	// MZU: 1 Zyklus verzögert M-Funktion 186
"MX_1Zykl_M187"	M 143.1	BOOL	// MZU: 1 Zyklus verzögert M-Funktion 187
"MX_1Zykl_M188"	M 143.2	BOOL	// MZU: 1 Zyklus verzögert M-Funktion 188
"MX_1Zykl_M189"	M 143.3	BOOL	// MZU: 1 Zyklus verzögert M-Funktion 189
"O_WW_1GRF_SPI"	M 143.5	BOOL	// M-AUSGANG: Werkzeuggreifer drehen Richtung Spindel
"O_WW_1_Klappe_auf"	M 143.6	BOOL	// M-AUSGANG: Werkzeugwechsler Tuer oeffnen
"M_WZWV_Beweg"	M 143.7	BOOL	// WZW: Werkzeug-Rueckhalt in Bewegung
"O_WW_1_Klappe_zu"	M 146.0	BOOL	// M-AUSGANG: Werkzeugwechsler Tuer schliessen
"I_WW_1GRF_MAG"	M 146.1	BOOL	// M-EINGANG: Werkzeuggreifer 1 Grundstellung Werkzeugmagazin
"I_WW_1GRF_SPI"	M 146.2	BOOL	// M-EINGANG: Werkzeuggreifer 1 Stellung Fraesspindel
"I_WW_1_Klappe_auf"	M 146.3	BOOL	// M-EINGANG: Werkzeugwechsler Tuer geoeffnet
"M_IMP_Asup_Init"	M 146.4	BOOL	// ASUP MACHINE: Initialisieren Flanke positiv
"M_FN_MANWZW"	M 146.6	BOOL	// WZW: Prozess / Manueller Wechsel aktiv Flanke negativ
"I_U_AXIS_MAIN_SW_ON"	M 146.7	BOOL	// M-EINGANG:
"M_WZW_VORG_AUSWERTUNG"	M 147.0	BOOL	// WZV: OMRON Regal Werkzeugwechsel Vorgewählt XXX
"M_Req_SPI_DATA"	M 147.2	BOOL	// VIBRATIONSSENSOR: Anforderung Spindeldaten lesen
"M_Sperre_TBef_FB193"	M 147.5	BOOL	// WZW: Nächsten T-Befehl sperren
"M_WZW_SPERRE_TBEF_V_MAG"	M 147.6	BOOL	// WZW: Sperre T-Befehl von MAG (Verfahren von Hand / Magazintüre offen)
"I_D_SF_NEG_PUMPE_EIN"	M 148.0	BOOL	// M-EINGANG: Diagnose Hebepumpe ein
"I_D_SF_NEG_PUMPE_AUS"	M 148.1	BOOL	// M-EINGANG: Diagnose Hebepumpe aus
"I_D_SF_NEG_UEBERLAUF"	M 148.2	BOOL	// M-EINGANG: Diagnose Hebepumpe Spaenefoerderer Not-Aus
"I_SF_PUMPE_EIN"	M 148.3	BOOL	// M-EINGANG: Hebepumpe Spaenefoerderer ein
"I_SF_PUMPE_AUS"	M 148.4	BOOL	// M-EINGANG: Hebepumpe Spaenefoerderer aus
"O_SF_PUMPE_EIN"	M 148.5	BOOL	// M-AUSGANG: Foerderpumpe Kuehlmittel ein
"I_KM_VOR_MIN_NIVEAU"	M 148.6	BOOL	// M-EINGANG: Kuehlmittel Vorwarnung Feinbereich Minimum
"I_KM_MIN_MAX_NIVEAU"	M 148.7	BOOL	// M-EINGANG: Kuehlmittel Niveaukontrolle Feinbereich
"I_KM_MAX_NIVEAU"	M 150.0	BOOL	// M-EINGANG: Kuehlmittel Fuellstand Maximum
"O_WZB_WB2_REINIGEN"	M 150.1	BOOL	// M-AUSGANG: Blasluft Werkzeugbruchueberwachung
"I_SF_SCHALTER_LINKS"	M 150.2	BOOL	// M-EINGANG: Spaenefoerderer Linkslauf
"O_SF_Linkslauf"	M 150.3	BOOL	// M-AUSGANG: Linkslauf Spaenefoerderer
"I_KM_MIN_VOR_NIVEAU"	M 150.4	BOOL	// M-EINGANG: Kuehlmittel Warnung Fuellstand Minimum
"I_KM_MIN_NIVEAU"	M 150.5	BOOL	// M-EINGANG: M-EINGANG: Kuehlmittel Fuellstand Minimum
"I_D_KM_MIN_NIVEAU"	M 150.6	BOOL	// M-EINGANG: Kuehlmittel Diagnose Fuellstand Minimum
"I_D_KM_MIN_VOR_NIVEAU"	M 150.7	BOOL	// M-EINGANG: Kuehlmittel Diagnose Warnung Minimum
"M_WZBR_WR"	M 152.0	BOOL	// WZW: Umschreiben OEM-Datum Werkzeugbruchüberwachung
"M_FP_WZBR_WR"	M 152.1	BOOL	// WZW: Umschreiben OEM-Datum Werkzeugbruchüberwachung FP
"override schreiben"	M 152.2	BOOL	// AX4: (C-Achse) Override schreiben Flanke positiv
"MX_ASpdl_RestwegLoeschen"	M 152.3	BOOL	// AX4: (C-Achse) Restweg löschen
"I_A_KM_TPF_MOTOR_EIN"	M 152.5	BOOL	// M-EINGANG: Kuehlmittel Diagnose Fuellstand Filtermulde
"M_BHG_PF_deaktiviert"	M 152.6	BOOL	// BHG: BHG deaktiviert Flanke positiv
"M_FN_KMTL_1"	M 152.7	BOOL	// KM: Kühlmittel 1 angewählt in Werkzeugliste Flanke negativ
"M_SpindleHold"	M 153.0	BOOL	// MSST: MCP IFM2 (Variant small) Spindel Halt
"M_SpindleDir"	M 153.1	BOOL	// MSST: MCP IFM2 (Variant small) Spindel drehen rechts(0) / links(1)
"M_FeedHold_from_FC24"	M 153.2	BOOL	// MSST: MCP IFM2 (Variant small) Vorschubsperre
"M_HM_PF_MBHG"	M 153.4	BOOL	// MBHG: Hilfsmerker positive Flanke
"M_HM_NF_MBHG"	M 153.5	BOOL	// MBHG: Hilfsmerker negative Flanke
"M_Anwahl_MBHG"	M 153.6	BOOL	// MBHG: Mini Bedienhangerät angewählt
"M_FP_INC_Abwahl"	M 153.7	BOOL	// BHG: Handrad bereit Flanke negativ -> Umschalltung JOG Dauerbetrieb
"M_BHG_Mag_links"	M 154.0	BOOL	// BHG: Magazin verfahren links
"M_BHG_Mag_rechts"	M 154.1	BOOL	// BHG: Magazin verfahren rechts
"M_pos_Fl_Tas_BHG_aktiv"	M 154.2	BOOL	// BHG: MSST Taste BHG aktivieren Flanke positiv
"M_an_abwaehl_BHG"	M 154.3	BOOL	// BHG: MSST Taste BHG aktivieren Impuls
"M_NCVar_lesen_Request"	M 154.7	BOOL	// SPINDEL:  Werkzeugdaten Istwert lesen (Request Get FB2)
"ReqFB198"	M 155.0	BOOL	// WZV: Anforderung Werkzeugdaten lesen
"M_Err_Rd_FB198"	M 155.1	BOOL	// WZV: Fehler Werkzeugdaten lesen
"M_Done_Rd_FB198"	M 155.2	BOOL	// WZV: Werkzeugdaten lesen fertig
"M_Wink_kopf_angewaehlt"	M 155.3	BOOL	// WZV: Winkelkopf in der Spindel
"M_WZ_Liste_Sp_rechts"	M 155.4	BOOL	// WZV: Spindel rechts angewählt in der Werkzeugliste
"M_WZ_Liste_SP_links"	M 155.5	BOOL	// WZV: Spindel links angewählt in der Werkzeugliste
"M_WZ_Liste_KM1"	M 155.6	BOOL	// WZV: Kühlmittel 1 angewählt in der Werkzeugliste
"M_WZ_Liste_KM2"	M 155.7	BOOL	// WZV: Kühlmittel 2  angewählt in der Werkzeugliste
"Mx_XAx_in_WZW_RAUM"	M 156.0	BOOL	// AX1: X-Achse im Werkzeugwechselraum
"M_WZ_Liste_Luftumsch."	M 156.1	BOOL	// WZV: Anwahl WZ-Liste (Shopmill) Wasser-Luft-Umschaltung
"M_FN_KMTL_2"	M 156.2	BOOL	// KM: Kühlmittel 2 angewählt in Werkzeugliste Flanke negativ
"M_FP_KM2_NCST"	M 156.4	BOOL	// KM: Kühlmittel 2 Nc-Start Flanke  positiv
"M_FP_KM1_NCST"	M 156.5	BOOL	// KM: Kühlmittel 1 Nc-Start Flanke  positiv
"M_FP_KM1_WZL"	M 156.6	BOOL	// WZV: Kühlmittel 1 angewählt in der Werkzeugliste Flanke positiv
"M_FP_KM2_WZL"	M 156.7	BOOL	// WZV: Kühlmittel 2 angewählt in der Werkzeugliste Flanke positiv
"M_Tool_Nr_geaendert"	M 157.0	BOOL	// SPINDEL:  Werkzeugnummer hat sich geaendert Impuls
"M_NCVar_lesen_Ready"	M 157.1	BOOL	// SPINDEL:  Werkzeugdaten Istwert lesen ready (Request Get FB2)
"M_FN_WZW_RESET"	M 157.2	BOOL	// OEM: Taste für Werkzeugwechsler rücksetzen Flanke negativ
"M_NC_Start_Prg_Anwahl"	M 157.4	BOOL	// STA: NC Start nach Programmanwahl
"M_OEM_IKZ_GESP"	M 158.0	BOOL	// OEM: Inneres Kühlmittel wird über Oem gesperrt
"O_FDSchmierung"	M 158.1	BOOL	// FRÄS-DREHTISCH SCHMIERUNG: einschalten
"M_KM_unterdruecken"	M 158.2	BOOL	// KM: Kühlmittel unterdrücken
"MX_IKZ_OVR_0"	M 158.3	BOOL	// KM: Vorschub-Override = 0 bei IKZ angewählt
"I_AL_HYD_FUELL_MIN_OK"	M 158.7	BOOL	// M-EINGANG: Fuellstand Hydraulik Minimum
"M_Sp_in_M19Pos"	M 159.0	BOOL	// AX6: Spindel in Werkzeugwechselposition
"I_D_KM_MAX_NIVEAU"	M 159.1	BOOL	// M-EINGANG: Kuehlmittel Diagnose Fuellstand Maximum
"I_KM_BTB_PNOZ"	M 159.2	BOOL	// M-EINGANG: Freigabe Kuehlmittelanlage PNOZ Not-Aus
"I_KM_BTB_ALLE_PUMPEN"	M 159.3	BOOL	// M-EINGANG: Freigabe Kuehlmittelanlage PNOZ Kabinentuer geschlossen
"I_KM_KRATZER_EIN"	M 159.4	BOOL	// M-EINGANG: Feinbereich Fuellstand Regeneration
"I_D_KM_KRATZER_EIN"	M 159.5	BOOL	// M-EINGANG: Diagnose Feinbereich Regeneration
"M_FP_KMTLUM_NCST"	M 159.6	BOOL	// KM: Kühlmittel Umschaltung Wasser/Luft Nc-Start Flanke  positiv
"M_FP_KMTL_UM"	M 159.7	BOOL	// KM: Kühlmittel Umschaltung Wasser/Luft Flanke  positiv
"M_MAG_Anforderung"	M 160.0	BOOL	// MAG: Magazinanforderung
"M_MAG_Fertig"	M 160.1	BOOL	// MAG: Magazinverfahren Fertig
"M_MAG_Start"	M 160.2	BOOL	// MAG: Magazinverfahren Start
"M_MAG_Laeuft"	M 160.3	BOOL	// MAG: Magazin Laeuft
"M_MAG_Fehler"	M 160.4	BOOL	// MAG: Magazin Fehler
"M_MAG_Stop"	M 160.5	BOOL	// MAG: Magazin Stop
"M_MAG_Freigabe"	M 160.6	BOOL	// MAG: Magazin Freigabe
"M_MAG_Links_Fahren"	M 160.7	BOOL	// MAG: Magazin Links
"M_MAG_Rechts_Fahren"	M 161.0	BOOL	// MAG: Magazin Rechts
"M_MAG_Ref_Gefunden"	M 161.1	BOOL	// MAG: Magazin Referenzpunkt gefunden
"M_MAG_Trigg_Ref_Gefunden"	M 161.2	BOOL	// MAG: Trigger Referenzpunkt gefunden
"M_MAG_Trigg_Tuer_Ver"	M 161.3	BOOL	// MAG: Trigger Tuer Verriegelt
"M_MAG_Trigg_SKR"	M 161.4	BOOL	// MAG: Trigger Softkey Rettung
"M_MAG_In_Position"	M 161.5	BOOL	// MAG: Magazin in Position
"M_MAG_Manuell_Rechts"	M 161.6	BOOL	// MAG: Magazin manuell Rechts
"M_MAG_Manuell_Links"	M 161.7	BOOL	// MAG: Magazin manuell Links
"M_WZW_Grdst"	M 170.0	BOOL	// WZW: Grundstellung
"I_KM_FEINB_MIN"	M 170.1	BOOL	// M-EINGANG: Feinbereich Fuellstand Minimum
"M_WZW_Aktiv"	M 170.2	BOOL	// WZW: Aktiver Ablauf
"M_WZW_Err"	M 170.3	BOOL	// WZW: Fehler
"M_WZW_Stat"	M 170.4	BOOL	// WZW: Statusfehler
"I_D_KM_FEINB_MIN"	M 170.5	BOOL	// M-EINGANG: Diagnose Feinbereich Minimum
"M_WZW_Hub_Beweg"	M 170.6	BOOL	// WZW: Hub in Bewegung
"M_WZW_Gre1_Mag_req"	M 171.0	BOOL	// WZW: Befehl Greifer 1 zum Magazin
"M_WZW_Greifer_OK"	M 171.1	BOOL	// WZW: Greifer OK (in Position Magazin oder Spindel)
"I_KM_FEINSTB_EIN"	M 171.2	BOOL	// M-EINGANG: Kuehlmittel Feinstbereich Fuellstand Minimum -> Pumpe Ein
"M_WZB_Anforderung"	M 171.3	BOOL	// WZB: WZ-Bruchüberwachung Ablauf starten
"M_WZB_Messung"	M 171.4	BOOL	// WZB: WZ-Bruchüberwachung Anforderung 2.Messung
"M_WZB_Ready"	M 171.5	BOOL	// WZB: WZ-Bruchüberwachung Rückmeldung
"M_WZW_Vorber_laeuft"	M 171.6	BOOL	// WZW: WZ-Vorbereitung läuft
"M_WZW_Gre1_Spi_req"	M 171.7	BOOL	// WZW: Befehl Greifer 1 zur Spindel
"MX_Vorschubsperre_Ax4"	M 173.0	BOOL	// AX4: (C-Achse) Vorschubsperre
"MX_RefPkt_4Achse"	M 173.1	BOOL	// AX4: (C-Achse) Referenzpunkt Achse
"MX_ASpdl_KorrWirksam"	M 173.2	BOOL	// AX4: (C-Achse) Vorschubkorrektur wirksam setzen
"MX_ASpdl_Spdl_Reset"	M 173.3	BOOL	// AX4: (C-Achse) Spindel Reset
"MX_ASpdl_Neu_Referenz"	M 173.4	BOOL	// AX4: (C-Achse) neu Referieren
"MX_ASpdl_Bei_Pos_NeuRef"	M 173.5	BOOL	// AX4: (C-Achse) bei Positionieren neu Referieren
"MX_ASpdl_GetrUmsch_82x3"	M 173.6	BOOL	// AX4: (C-Achse) Getriebeumschaltung 82x3
"MX_ASpdl_PosBetr_84x5"	M 173.7	BOOL	// AX4: (C-Achse) Positionierbetrieb
"I_WW_1_ZYL_SPI"	M 175.0	BOOL	// M-EINGANG: Werkzeugmagazin Stellung Spindel
"I_WM_WZ_ZYL_CLAMP"	M 175.1	BOOL	// M-EINGANG: Pneumatikzylinder Werkzeug loesen eingefahren Grundstellung
"I_WM_WZ_ZYL_RELEASE"	M 175.2	BOOL	// M-EINGANG: Pneumatikzylinder Werkzeug loesen ausgefahren
"I_WM_WZ_SPI_CLAMP"	M 175.3	BOOL	// M-EINGANG: Werkzeug verriegelt Wechselposition
"I_WM_WZ_RPL_CLAMP"	M 175.4	BOOL	// M-EINGANG: Werkzeug verriegelt Werkzeugeingabestation
"I_WM_WZ_MAN_Relase"	M 175.5	BOOL	// M-EINGANG: Werkzeug manuell lösen
"I_WM_WZ_MAN_CLAMP"	M 175.6	BOOL	// M-EINGANG: Werkzeug manuell klemmen
"M_NewTool_Grf2"	M 176.0	BOOL	// WZV: Neues Werkzeug für Greifer 2
"M_SpTool_Grf2"	M 176.1	BOOL	// WZV: Spindelwerkzeug für Greifer 2
"M_NewTool_WFK"	M 176.2	BOOL	// WZV: Neues Werkzeug Winkelfräskopf
"M_SpWZ_WFK"	M 176.3	BOOL	// WZV: Spindelwerkzeug Winkelfräskopf
"I_PW_PNOZ_FREIGABE"	M 176.4	BOOL	// M-EINGANG: Freigabe von PNOZ für Palettenwechsler
"M_TI_WZ_BEZEICHNER"	M 176.5	BOOL	// WZVS mit MCU Werkzeugbezeichner
"M_FP_RPL_Tuere_auf"	M 176.6	BOOL
"M_FP_Kabine_auf"	M 176.7	BOOL
"MX_ASpdl_DrehGrenz_83x0"	M 177.0	BOOL	// AX4: (C-Achse) Drehzahlgrenze
"MX_ASpdl_GewBohnre_84x3"	M 177.1	BOOL	// AX4: (C-Achse) Gewindebohren aktiv
"MX_ASpdl_SollBer_83x5"	M 177.2	BOOL	// AX4: (C-Achse) Spindel im Sollbereich
"MX_ASpdl_PendBetr_84x5"	M 177.3	BOOL	// AX4: (C-Achse) Pendelbetrieb
"MX_ASpdl_E_RUCompl_94x2_"	M 177.4	BOOL	// AX4: (C-Achse) Hochlauf beendet
"MX_ASpdl_Message_94x7"	M 177.5	BOOL	// AX4: (C-Achse) Variable Meldefunktion
"MX_ASpdl_A_RefVerz_12x7"	M 177.6	BOOL	// AX4: (C-Achse) Referenzverzögerung bei Motormessystem
"MX_ASpdl_M3"	M 177.7	BOOL	// AX4: (C-Achse) M3 (Rechtslauf) aktiv
"MX_ASpdl_M4"	M 178.0	BOOL	// AX4: (C-Achse) M4 (Linkslauf) aktiv
"MX_ASpdl_M5"	M 178.1	BOOL	// AX4: (C-Achse) M5 (Aus) aktiv
"MX_ASpdl_M3_M4"	M 178.2	BOOL	// AX4: (C-Achse) M3 oder M4 oder Fahrbefehl aktiv
"MX_ASpdl_IMP_M3"	M 178.3	BOOL	// AX4: (C-Achse) M3 (Rechtslauf) aktiv Impuls
"MX_ASpdl_IMP_M4"	M 178.4	BOOL	// AX4: (C-Achse) M4 (Linkslauf) aktiv Impuls
"MX_ASpdl_IMP_M5"	M 178.5	BOOL	// AX4: (C-Achse) M5 (Aus) aktiv Impuls
"MX_ASpdl_IMP_M3_M4"	M 178.6	BOOL	// AX4: (C-Achse) M3 oder M4 Impuls
"MX_ASpdl_Reset_M3_4"	M 178.7	BOOL	// AX4: (C-Achse) Reset M3 oder M4
"MX_WZW_Langsam_Ein"	M 179.0	BOOL	// WZW: Werkzeugwechsel Einwechseln langsam
"MX_WZW_Langsam_Aus"	M 179.1	BOOL	// WZW: Werkzeugwechsel Auswechseln langsam
"MX_WZW_Langsam_Voll"	M 179.2	BOOL	// WZW: Werkzeugwechsel Vollwechsel langsam
"m_179.3"	M 179.3	BOOL	// Reserve
"M_WZW_Reset_Module"	M 179.4	BOOL	// WZW: Reset aller Module des WZW
"m_179.5"	M 179.5	BOOL	// Reserve
"M_WZW_Reset"	M 179.6	BOOL	// WZW: Reset steht an
"M_TR_Freigabe_PW"	M 179.7	BOOL	// PW: Freigabe Palettenwechsler Flanke positiv
"M_PW_Status"	M 180.0	BOOL	// PW: Stop aus Statusueberwachung
"M_PW_Err"	M 180.1	BOOL	// PW: Fehler Palettenwechlser
"I_D_KM_FEINSTB_EIN"	M 180.2	BOOL	// M-EINGANG: Kuehlmittel Diagnose Feinstbereich Minimum
"M_FreigabePW"	M 180.3	BOOL	// PW: Freigabe Palettenwechsler
"I_KM_FEINSTB_AUS"	M 180.4	BOOL	// M-EINGANG: Kuehlmittel Feinstbereich Fuellstand Maximum
"I_D_KM_FEINSTB_AUS"	M 180.5	BOOL	// M-EINGANG: Kuehlmittel Diagnose Feinstbereich Maximum
"I_KM_FEINSTB_MIN"	M 180.6	BOOL	// M-EINGANG: Kuehlmittel Feinstbereich Fuellstand Grenzwertmeldung
"I_D_KM_FEINSTB_MIN"	M 180.7	BOOL	// M-EINGANG: Kuehlmittel Diagnose Feinstbereich Grenzwertmeldung
"I_KM_DRUCK2_M7_EIN"	M 181.0	BOOL	// M-EINGANG: Kuehlmittel Freigabe Maschine Druckstufe 2
"M_Sp_inM19PosWFK"	M 181.1	BOOL	// AX6: Spindel in Position Winkelfräskopfposition
"m_181.2"	M 181.2	BOOL	// Reserve
"M_FN_PW_Hub_unten"	M 181.3	BOOL	// PW: Palettenwechler Hub unten Flanke negativ
"M_FP_PW_Hub_unten"	M 181.4	BOOL	// PW: Palettenwechler Hub unten Flanke positiv
"M_Stange_Aktiv"	M 181.6	BOOL	// STA: Stange aktiv
"M_PW_Aktiv"	M 181.7	BOOL	// PW: Wechsel aktiv
"M_PW_GRDST"	M 182.0	BOOL	// PW: Wechsler in Grundstellung
"M_PW_Reset"	M 182.1	BOOL	// PW: Reset Merker
"m_182.2"	M 182.2	BOOL	// Reserve
"M_TR_Start_PW"	M 182.3	BOOL	// PW: Trigger Start PW
"M_FP_Resettaste"	M 182.4	BOOL	// PW Taste Reset Flanle positiv
"M_TR_Ende_PW"	M 182.5	BOOL	// PW: Trigger Ende PW
"m_182.6"	M 182.6	BOOL	// Reserve
"M_PW_Pal_Vorhanden"	M 182.7	BOOL	// PW: Palette vorhanden
"m_183.0"	M 183.0	BOOL	// Reserve
"m_183.1"	M 183.1	BOOL	// Reserve
"m_183.2"	M 183.2	BOOL	// Reserve
"m_183.3"	M 183.3	BOOL	// Reserve
"m_183.4"	M 183.4	BOOL	// Reserve
"M_MD_lesen_Hochlauf"	M 183.5	BOOL	// PLC NCK: Maschinendaten beim Hochlauf lesen
"Mx_MT_KAL_Klappe_zu"	M 183.6	BOOL	// Merker Schmutzklappe Kalibriereinrichtung geschlossen
"M_FP_BildAnwahl"	M 183.7	BOOL	// MA: Bild für Wuchten aufrufen Flanke positiv
"MX_H5020"	M 184.0	BOOL	// WZW: H-Funktion 5020 Start Werkzeugwechslerklappe öffnen
"MX_H5021"	M 184.1	BOOL	// WZW: H-Funktion 5021 Start Werkzeugwechslerklappe schliesen
"M_LASER_AKTIV_FP"	M 184.2	BOOL	// LASER: Laser aktiv Flanke positiv
"I_D_KM_MIN_MAX_NIVEAU"	M 184.3	BOOL	// M-EINGANG: Kuehlmittel Diagnose Niveaukontrolle Feinbereich
"Mx_LA_Klappe_zu"	M 184.4	BOOL	// Merker Schmutzblende geschlossen
"I_D_KM_VOR_MIN_NIVEAU"	M 184.5	BOOL	// M-EINGANG: Kuehlmittel Diagnose Vorwarnung Feinbereich
"MX_PW_HUB_VOR_MITTE_HEBE"	M 184.6	BOOL	// PW: Hub vor Mitte heben Impuls
"MX_PW_HUB_VOR_MITTE_SENK"	M 184.7	BOOL	// PW: Hub vor Mitte senken Impuls
"Mx_H5010"	M 186.0	BOOL	// WZW: H-Funktion 5010 Hub zur Spindelstellung
"Mx_H5011"	M 186.1	BOOL	// WZW: H-Funktion 5011 Hub zur Grundstellung
"m_186.2"	M 186.2	BOOL	// Reserve
"M_IBN_Handlingsystem"	M 186.3	BOOL	// IBN: Handlinsystem
"M_PW_SpV_Zu_Bew"	M 186.4	BOOL	// PW: Spannvorrichtung klemmen
"M_PW_Klemm_Bew"	M 186.5	BOOL	// PW: Klemmung in Bewegung
"M_PW_HubMitte_Bew"	M 186.6	BOOL	// PW: Hub zur Mitte Bewegung
"M_PW_HubUnten_Bew"	M 186.7	BOOL	// PW: Hub Unten Bewegung
"M_PW_HubOben_Bew"	M 187.0	BOOL	// PW: Hub Oben Bewegung
"M_PW_Dreh_Bew"	M 187.1	BOOL	// PW: Dreh - Bewegung
"O_KM_Motor_Kratzfoerd"	M 187.2	BOOL	// M-AUSGANG: Antrieb Kratzerfoerderer
"M_PW_Zeitschmierung_ein"	M 187.3	BOOL	// PW-Schmierung: Zeitschmierung ein
"M_WZW_Ausw"	M 187.4	BOOL	// WZW: WZ-Ablegevorgang
"M_WZW_Gre1_Keg_req"	M 187.5	BOOL	// WZW: Greifer 1 zur Kegelreinigung
"M_WZW_Gre2_Keg_req"	M 187.6	BOOL	// WZW: Greifer 2 zur Kegelreinigung
"O_KM_PUMPE_FILTER_FEINB"	M 187.7	BOOL	// M-AUSGANG: Foerderpumpe Feinstbereich
"M_Req_externe_NV"	M 188.0	BOOL	// Anforderung Anwahl externe Nullpunktverschiebung
"M_Error_externe_NV"	M 188.1	BOOL	// Fehler beim Schreiben der externen Nullpunktverschiebung
"M_FP_Req_externe_NV"	M 188.2	BOOL	// Anforderung Anwahl externe Nullpunktverschiebung Flanke positiv
"M_FP_PW_FREIGABE"	M 188.3	BOOL	// Bedingungen für Rohteil setzen Flanke positiv
"m_VSH_SP_WZ_NIO"	M 188.4	BOOL
"m_M3_M4_aktiv"	M 188.5	BOOL
"M_FI_WW_POS_FRG_WZM"	M 188.6	BOOL	// WZW: Fehler Eingang Freigabe Magazin
"M_WZW_Gre1_Pos_Mag"	M 189.0	BOOL	// WZW: Greifer 1 Position Magazin
"M_WZW_Gre1_Pos_Spi"	M 189.1	BOOL	// WZW: Greifer 1 Position Spindel
"M_WZW_Gre1_Pos_Keg"	M 189.2	BOOL	// WZW: Greifer 1 Position Kegelreinigung
"M_WZW_Gre2_Pos_Keg"	M 189.3	BOOL	// WZW: Greifer 2 Position Kegelreinigung
"M_WZW_Hub_Mag_req"	M 189.4	BOOL	// WZW: Befehl Hub zum Magazin
"M_WZW_Hub_GrdSt_req"	M 189.5	BOOL	// WZW: Befehl Hub in Grundstellung
"M_WZWV_Grundstell_req"	M 189.6	BOOL	// WZW: Befehl Werkzeug-Rueckhalt zur Grundstellung
"M_WZWV_Verrieg_req"	M 189.7	BOOL	// WZW: Befehl Werkzeug-Rueckhalt ausfahren (verriegeln)
"M_WSP_in_Bewegung"	M 190.0	BOOL	// WSP: Werkzeugspanner in Bewegung
"M_WZSP_entprellt"	M 190.1	BOOL	// WSP: Werkzeugspanner ist entprellt
"M_WZSP_Trigger_oeffnen"	M 190.2	BOOL	// WSP: Werkzeugspanner oeffnen Trigger
"M_WZSP_Trigger_schliess"	M 190.3	BOOL	// WSP: Werkzeugspanner schliessenTrigger
"M_WZSP_Timer_Start"	M 190.5	BOOL	// WSP: Startbit zum Anstoss von Verzoegerungszeit
"m_WZ_entladen_67015"	M 190.6	BOOL	// Werkzeugentladen Fehler 67015
"m_WZ_entladen_67027"	M 190.7	BOOL	// Werkzeugentladen Fehler 67027
"I_WW_ZYL1_FRG_MAG"	M 191.0	BOOL	// M-EINGANG: Freigabe drehen Werkzeugmagazin
"M_WZSP_Trigg1"	M 191.2	BOOL	// WSP: Trigger Werkzeugspanner
"M_WZSP_angewaehlt"	M 191.3	BOOL	// WSP: Werkzeugspanner angewaehlt
"M_WZSP_Verriegelung"	M 191.5	BOOL	// WSP: Werkzeugspanner-Verriegelung Spindel
"M_WZSP_Zeit_nach_NotAus"	M 191.7	BOOL	// WSP: Zeit nach Not-Aus abgelaufen
"M_WZSP_Spindel_sperren"	M 195.0	BOOL	// WSP: Spindel durch Werkzeugspanner gesperrt
"M_WZ_Spanner_Auf"	M 195.1	BOOL	// WSP: Spanner auf
"M_WZ_Spanner_Zu"	M 195.2	BOOL	// WSP: Spanner Zu
"M_Man_WZSP_Auf"	M 195.3	BOOL	// WSP: Anforderung Manuelles Spanner loesen
"M_Auto_WZSP_Auf"	M 195.4	BOOL	// WSP: Anforderung Automatisches Spanner loesen
"M_O_Anwahl_WZS_Man"	M 195.5	BOOL	// WSP: Ausgang Manuelles loesen Spanner
"M_Umsp_Aus_Spindel"	M 195.6	BOOL	// WZV: Umspeichern WZ aus Spindel
"M_Umsp_in_Spindel"	M 195.7	BOOL	// WZV: Umspeichern WZ in Spindel
"M_H5001_WW_Ende"	M 197.0	BOOL	// WZW: H-Funktion 5001 Werkzeugwechsel beendet
"M_H5003_Wz_spannen"	M 197.1	BOOL	// WZW: H-Funktion 5003 Werkzeugspanner in Spindel schliessen
"M_H5008_DT_Sp_Mag"	M 197.2	BOOL	// WZW: H-Funktion 5003 Datentausch Spindel > Magazin
"M_H5007_H5009_DT_Mag_Sp"	M 197.3	BOOL	// WZW: H-Funktion 5007 / 5009 Datentausch Magazin > Spindel / Spanner zu
"I_WZSP_gespannt_oWZ"	M 197.4	BOOL	// M-EINGANG: Werkzeugspanner gespannt ohne Werkzeug
"M_Spindel_leer"	M 197.5	BOOL	// WZW Teller: Spindel leer
"O_WM_WZ_STAT_einlegen"	M 197.6	BOOL	// M-AUSGANG: WZV: Lampe TIN (Werkzeug einlegen)
"O_WM_WZ_STAT_entnehmen"	M 197.7	BOOL	// M-AUSGANG: WZV: Lampe TOUT  (Werkzeug entnehmen)
"M_Fehler_WZSpanner"	M 199.0	BOOL	// WSP: Fehler im Werkzeugspanner
"M_WZSP_Trigg"	M 199.1	BOOL	// WSP: Trigger Move
"M_WZSP0_Move"	M 199.2	BOOL	// WSP: Bewegung Spannertyp 0
"M_WZSP_Trigg_TuerZu"	M 199.3	BOOL	// WSP: Trigger Tuer zu
"FP_I_WM_Beladung_zu"	M 199.4	BOOL	// WZV: Beldadung zu Flanke positiv
"M_WZV_T-Daten_req"	M 199.5	BOOL	// WZV: Daten aus T-Befehl falsch
"M_WZV_REQ_Data"	M 199.6	BOOL	// WZV:Request Werkzeugdaten lesen
"M_WZV_Positionieren_S"	M 199.7	BOOL	// WZV: Positionieren beendet (gespeichert)
"ASUP_Machine_active"	M 201.0	BOOL	// ASUP-fc201 ASUP_MACHINE  aktiv
"Start_ASUP_Machine_Nr.1"	M 201.1	BOOL	// ASUP-fc201 1 Werkzeugwechsler Rettung (Einrichten)
"Start_ASUP_Machine_Nr.2"	M 201.2	BOOL	// ASUP-fc201 2 Palettenwechslerwechsler Rettung (Einrichten)
"Start_ASUP_Machine_Nr.3"	M 201.3	BOOL	// ASUP-fc201 3 Nach Hochlauf und Referieren den Fahrbereich M56 aktivieren
"Start_ASUP_Machine_Nr.4"	M 201.4	BOOL	// ASUP-fc201 4
"Start_ASUP_Machine_Nr.5"	M 201.5	BOOL	// ASUP-fc201 5 Temperaturkompensation Ein
"Start_ASUP_Machine_Nr.6"	M 201.6	BOOL	// ASUP-fc201 6  Werkzeugdaten ins DPR lesen
"Start_ASUP_Machine_Nr.7"	M 201.7	BOOL	// ASUP-fc201 7 Winkelfräßkopf Rettung (Einrichten)
"ASUP_Frame_active"	M 203.0	BOOL	// ASUP-fc203 ASUP_FRAME aktiv
"M_ASUP_Trafo_ON"	M 203.1	BOOL	// ASUP-fc203 1
"Start_ASUP_Frame_Nr.2"	M 203.2	BOOL	// ASUP-fc203 2
"M_ASUP_INIT_READY"	M 205.0	BOOL	// ASUP-Initialisierung Fertig
"M_KM_Anlage_angewaehlt"	M 205.1	BOOL	// KM: Maschinenparameter Kühlmittelanlage angewählt
"M_RESET_DURCH_RS_HS"	M 205.3	BOOL	// WZV: Reset durch Rundspeicher / Handlingsystem bei WZ-Bruch
"M_RESET_WZV"	M 205.4	BOOL	// WZV: Reset-Taste für Werkzeugverwaltung
"M_RESET_DISABLE"	M 205.5	BOOL	// WZV: Reset verzögern für WZV
"M_FN_Reset_WZV"	M 205.6	BOOL	// WZV: Reset WZV Flanke negativ
"O_SP_MPL_BLASLUFT"	M 205.7	BOOL	// M-AUSGANG: Blasluft Medienkupplung Spannhydraulik 'Ein'
"M_INIT_ASUP_Maschine"	M 206.0	BOOL	// ASUP Init Asup Maschine
"M_INIT_ASUP_Frame"	M 206.2	BOOL	// ASUP Init Asup Frame
"MX_1Job_Maschine"	M 206.3	BOOL
"M_FP_start_up_shopmill"	M 206.5	BOOL	// SHOPMILL: Startup Flanke positiv
"M_Temp"	M 206.6	BOOL	// SHOPMILL: Window ausblenden wenn Shopmill geladen wird
"M_FP_shopmill_activ"	M 206.7	BOOL	// SHOPMILL: Application aktiv Flanke positiv
"I_AL_BTB_PNOZ"	M 208.0	BOOL	// M-EINGANG: Betriebsbereit Sicherheitsschaltgeraet
"M_tds_lesen_last_part"	M 208.1	BOOL	// TDS: BALLUFF Werkzeugdaten lesen last part
"M_tds_write_last_part"	M 208.2	BOOL	// TDS: BALLUFF Werkzeugdaten schreiben last part
"M_TDS_vgl"	M 208.3	BOOL	// TDS: BALLUFF Werkzeugdaten Vergleich
"M_TDS_BALLUFF_aktiv"	M 208.4	BOOL	// TDS für Balluff ist aktiv
"M_TDS_BILZ_aktiv"	M 208.5	BOOL	// TDS für BILZ ist aktiv
"M_FP_Kanal_Reset"	M 209.0	BOOL	// Impuls Reset Taster
"M_Verfahrbefehl_steht_an"	M 210.0	BOOL	// MA: Verfahrbefehl steht an
"M_pos_Flanke_M30"	M 210.1	BOOL	// MA: Kanal 1 M30 Flanke positiv
"M_M30_Kanal1"	M 210.2	BOOL	// MA: Kanal1 M30 wurde ausgeloest
"M_FP_NCStart_Warmlpr"	M 210.3	BOOL	// MA: Warmlaufprogramm NC Start Flanke positiv
"M_Imp_NCStart"	M 210.4	BOOL	// MA: Warmlaufprogramm NC Start Impuls
"M_NC_Start_Warmlpr"	M 210.6	BOOL	// MA: Warmlaufprogramm NC Start
"M_pos_Fl_BHG_angewaehlt"	M 214.0	BOOL	// BHG: BHG angewaehlt Flanke positiv
"M_neg_Fl_BHG_angewaehlt"	M 214.1	BOOL	// BHG: BHG angewaehlt Flanke negativ
"M_5te_6te_BHG"	M 214.2	BOOL	// BHG: Achse 5 oder Spindel auf + - Taste, vor Anwahl BHG
"M_24aktiv"	M 214.3	BOOL	// LA: Laser ausfahren M24 aktiv
"Mx_Sperre_BAchse"	M 214.4	BOOL	// AX: Verfahrbereiche -> Sperre B-Achse
"M_Blum_Flanke1"	M 214.5	BOOL	// LA:  FC_ZYLINDER Flanke 1
"M_Blum_Laser_Ausgef"	M 214.7	BOOL	// LA:  Laser ausgefahren
"M_Warm_Fkt_FN_aktiv"	M 215.0	BOOL	// PW: Warmlauffunktion aktiv Flanke negativ
"M_Warm_Fkt__FP_aktiv"	M 215.1	BOOL	// PW: Warmlauffunktion aktiv Flanke positiv
"O_PW_RPL_OFFEN"	M 215.2	BOOL	// PW: Ruestplatztür offen
"O_ROBOT_FREIGABE"	M 215.3	BOOL	// ROBOT: Freigabe Werkstueckwechsel Handlingsystem
"O_ROBOT_START"	M 215.4	BOOL	// ROBOT: Startsignal Werkstueckwechsel Handlingsystem
"M_FN_PW_AKTIV"	M 215.5	BOOL	// HM neg.Flanke PW_AKTIV
"O_ROBOT_AUTO_BELADEN"	M 215.6	BOOL	// ROBOT: Betriebsart automatisch Beladen
"M_IMP_FN_PW_AKTIV"	M 215.7	BOOL	// Impuls neg.Flanke PW_AKTIV
"O_ROBOT_PALETTE2_180°"	M 216.1	BOOL	// ROBOT: Palettenwechsler Stelllung 180 Grad Palette 2
"M_Blum_Flanke2"	M 216.2	BOOL	// LA:  FC_ZYLINDER Flanke 2
"O_ROBOT_SPV_RPL_GELOEST"	M 216.3	BOOL	// ROBOT: Spannvorrichtung Ruestplatz geloest
"O_ROBOT_SPV_RPL_GESPANN"	M 216.4	BOOL	// ROBOT: Spannvorrichtung Ruestplatz gespannt
"I_SP_FILTER_WAR"	M 216.7	BOOL	// M-Eingang: FD-Spannhydraulik ohne PROP-Ventil Filter verschmutzt
"I_PW_AUTO_EIN_3R"	M 217.0	BOOL	// M-EINGANG: Automatik Werkstueckwechsel Ein
"I_PW_RP_GELOEST"	M 217.1	BOOL	// M-EINGANG: Paletten-Ruestplatz Klemmung geloest
"I_ROBOT_BELADEN_ENDE"	M 217.3	BOOL	// M-EINGANG: Rueckmeldung Werkstueckwechsel Handlingsystem
"M_Reset_WZW"	M 217.4	BOOL	// WZW: Reset Werkzeugwechsel
"M_FP_Not_aus"	M 217.5	BOOL	// WZW: Maschine Aus Flanke positiv
"MX_FP1_Wizzard"	M 217.6	BOOL	// WIZARD: Umschalten Kuehlmittel / Blasluft Flanke positiv
"MX_FP2_Wizzard"	M 217.7	BOOL	// WIZARD: Umschalten Kuehlmittel / Blasluft Flanke negativ
"M_SK_ERR"	M 224.0	BOOL	// SCHWENKKOPF:Fehlerbit
"M_FP_SK_Resettaste"	M 224.1	BOOL	// SCHWENKKOPF:Taste Reset Flanke positiv
"M_SK_Reset"	M 224.2	BOOL	// SCHWENKKOPF:Reset Merker
"M_SK_Reset_Module"	M 224.3	BOOL	// SCHWENKKOPF:Reset SK Module
"M_SK_Rett1"	M 224.4	BOOL	// SCHWENKKOPF:Status Rettungsbit 1
"M_SK_Rett2"	M 224.5	BOOL	// SCHWENKKOPF:Status Rettungsbit 2
"M_SK_Rett3"	M 224.6	BOOL	// SCHWENKKOPF:Status Rettungsbit 3
"M_SK_Rett4"	M 224.7	BOOL	// SCHWENKKOPF:Status Rettungsbit 4
"M_SK_Stat"	M 225.0	BOOL	// SCHWENKKOPF:Stop aus Statusueberwachung
"M_TR_Ende_SK"	M 225.1	BOOL	// SCHWENKKOPF:Trigger Ende SK
"M_TR_Start_SK"	M 225.2	BOOL	// SCHWENKKOPF:Trigger Start SK
"M_SK_Aktiv"	M 225.3	BOOL	// SCHWENKKOPF:Wechsel aktiv
"M_SK_GRDST"	M 225.4	BOOL	// SCHWENKKOPF:Schwenkkopf in Grundstellung
"M_SK_Klemm_Bewegung"	M 225.5	BOOL	// SCHWENKKOPF:Klemmung Bewegung steht an
"M_SK_Kopf_Bewegung"	M 225.6	BOOL	// SCHWENKKOPF:Kopf Bewegung steht an
"M_SK_TR_Ende_M26x"	M 225.7	BOOL	// SCHWENKKOPF:Trigger Ende M26x
"M_TR_Start_Suchlauf"	M 227.0	BOOL	// KM: Start Satzsuchlauf Flanke positiv
"M_FN_Maschine_ein"	M 227.2	BOOL	// MA: Flanke Negativ Maschine Ein HM
"M_FP_Maschin"	M 227.3	BOOL	// MA: Flanke Positiv Maschine Ein HM
"M_SK_FB1_aktiv"	M 227.4	BOOL	// SCHWENKKOPF:Fahrbereich 1 aktiv
"M_SK_FB2_aktiv"	M 227.5	BOOL	// SCHWENKKOPF:Fahrbereich 2 aktiv
"M_SK_FB3_aktiv"	M 227.6	BOOL	// SCHWENKKOPF:Fahrbereich 3 aktiv
"M_SK_Fahrbereich_gesamt"	M 227.7	BOOL	// SCHWENKKOPF:Fahrbereich ohne Einschränkung
"M_pos_Trigg_SKR_Taste"	M 231.0	BOOL	// SOFTKEYRETTUNG: Taste Flanke positiv
"M_neg_Trigg_SKR_Taste"	M 231.1	BOOL	// SOFTKEYRETTUNG: Taste Flanke negativ
"M_Flankenmerker_positiv"	M 231.2	BOOL	// SOFTKEYRETTUNG: Flanlenmerker
"M_4Ax_Messystem_direkt"	M 231.3	BOOL	// AX4: Achse 4 direktes Messystem
"M_5Ax_Messystem_direkt"	M 231.4	BOOL	// AX5: Achse 5 direktes Messystem
"M_wzw_pw_p_Flanke"	M 231.6	BOOL	// SOFTKEYRETTUNG: Maske PW oder WZW angewaehlt
"M_Anw_FP"	M 231.7	BOOL	// SOFTKEYRETTUNG: Anwender-Maske angewaehlt Flanke positiv
"M_WZ_anlegen"	M 232.0	BOOL
"NC_DATEN_LESEN_ENTLADEN"	M 232.1	BOOL
"M_Siro_db137"	M 232.2	BOOL
"M_RegGr_inGasse_aktiv"	M 233.0	BOOL	// WZW OMRON: Regalgreifer in Gasse aktiv
"M_RegGr_schliessen_aktiv"	M 233.1	BOOL	// WZW OMRON: Regalgreifer schliessen aktiv
"M_RegGr_auf_VP"	M 233.2	BOOL	// WZW OMRON: Regalgreifer in Vorposition
"M_RegGr_auf_WP"	M 233.3	BOOL	// WZW OMRON: Regalgreifer in Wechselposition
"M_FP_Quit_Kd9"	M 233.4	BOOL	// WZW OMRON: Quittierung Komando 9 Flanke positiv
"M_FP_Quit_Kd14"	M 233.5	BOOL	// WZW OMRON: Quittierung Komando14 Flanke positiv
"M_FP_Quit_Kd17"	M 233.6	BOOL	// WZW OMRON: Quittierung Komando 17 Flanke positiv
"M_FP_Quit_Kd16"	M 233.7	BOOL	// WZW OMRON: Quittierung Komando 16 Flanke positiv
"M_Sp_leeren aktiv"	M 234.0	BOOL	// WZW OMRON: Spindel leeren aktiv
"M_FP_Quit_Kd13"	M 234.1	BOOL	// WZW OMRON: Quittierung Komando 13 Flanke positiv
"M_RegGr_oeffnen_aktiv"	M 234.2	BOOL	// WZW OMRON: Regalgreifer öffnen aktiv
"M_RegGr_schliess_aktiv"	M 234.3	BOOL	// WZW OMRON: Regalgreifer schliessen aktiv
"MX_Hub_Mitte_von_oben"	M 234.4	BOOL	// PW: Hub Mitte von Oben
"MX_Hub_Mitte_von_unten"	M 234.5	BOOL	// PW: Hub Mitte von Unten
"MX_FP_Hub_Bewegung"	M 234.6	BOOL	// PW: Hub Bewegung Flanke positiv
"MX_Hub_Bewegung"	M 234.7	BOOL	// PW: Hub Bewegung Impuls
"HM_PI_RegGreifer_GRST"	M 235.2	BOOL	// WZW OMRON: HMI Regalgreifer zur Grundstellung
"HM_PI_WZ_aus_Spi"	M 235.3	BOOL	// WZW OMRON: HMI Werkzeug aus Spindel entnehmen
"M_RFG_Spindel_Wizard"	M 236.0	BOOL	// SPINDEL: Reglerfreigabe durch Wizard
"M_FP_Spi_RFG_Wizard"	M 236.1	BOOL	// SPINDEL: Reglerfreigabe durch Wizard Flanke positiv
"M_FP_Spi_inReg_Wizard"	M 236.2	BOOL	// SPINDEL: In Regelung Flanke positiv
"I_Spannfutter_Aachsgekl"	M 236.3	BOOL	// M-EINGANG: STA: Eingang Spannfutter geklemmt
"MX_FP_Hub_Mitte"	M 236.4	BOOL	// PW: Hub Mitte Flanke positiv
"MX_FN_Hub_Mitte"	M 236.5	BOOL	// PW: Hub Mitte Flanke negativ
"M_M97_M98_unterdrücken"	M 236.7	BOOL	// KM: M97 / M98 (Spänespülung / Werkstückspülung) unterdrücken
"MX_O_4Ax_loesen"	M 237.0	BOOL	// AX4: (C-Achse) Ausgang Klemmung lösen
"MX_Rundachsanf_aktiv"	M 237.1	BOOL	// AX: Rundachsmodul Anforderung aktiv
"M_SPP_ein_neg_Fl"	M 237.3	BOOL	// SPÄNESPÜLUNG: Ausgang Spülpistole Aus Flanke negativ
"Mx_Pal_Stoerung_WZBruch"	M 237.7	BOOL	// WZB: Störung Werkzeugbruch
"M_M11_aktiv"	M 238.0	BOOL	// AX: M-Funktion 11 (Klemmung Achse 4 lösen) aktiv
"MX_FP_Start_ASUP_1"	M 238.1	BOOL	// ASUP 1: Flanke für Start des ASUPs
"Mx_FP_pos_Trigg_Blau_KR"	M 239.0	BOOL	// Kalibrierring: FP_pos_Trigg_Blau
"Mx_FN_neg_Trigg_Blau_KR"	M 239.1	BOOL	// Kalibrierring: FN_neg_Trigg_Blau
"Mx_FP_pos_Trigg_Gelb_KR"	M 239.2	BOOL	// Kalibrierring: FP_pos_Trigg_Gelb
"Mx_FN_neg_Trigg_Gelb_KR"	M 239.3	BOOL	// Kalibrierring: FN_neg_Trigg_Gelb
"M_Kalibrier_Ring_Ausgef"	M 239.4	BOOL	// KR: Kalibrierring ausgefahren
"M_Kalibrierring_Flanke1"	M 239.5	BOOL	// Kalibriering:  FC_ZYLINDER Flanke 1
"M_Kalibrierring_Flanke2"	M 239.6	BOOL	// Kalibriering:  FC_ZYLINDER Flanke 2
"M_Umsch_5/6_Achse"	M 240.0	BOOL	// MSST: Handrad ein Flanke positiv
"MX_Verfahrbefehl"	M 240.1	BOOL	// MSST: Fahrbefehl Achstasten
"M_FP_MKS/WKS"	M 240.2	BOOL	// MSST: Umschaltung MKS/WKS Flanke positiv
"M_FP_Handrad_Ein"	M 240.3	BOOL	// MSST: Handrad ein Flanke positiv
"Mx_FP_wz_melden"	M 240.4	BOOL	// SINRPC: Werkzeug melden Flanke positiv
"M_MTaster_in_Spi"	M 240.7	BOOL	// MESSTASTER: Messtaster (WZ-Typ 710) in Spindel
"M_FP_Spi_In_Pos"	M 241.0	BOOL	// MESSTASTER: Flanke Spindel in Position
"MX_MTaster_Aktiv"	M 241.1	BOOL	// MESSTASTER: Taster aktiv
"MX_Flanke_MT_Ein"	M 241.2	BOOL	// MESSTASTER: Flanke MT ein
"MX_MT_Flanke_MT_Aus"	M 241.3	BOOL	// MESSTASTER: Flanke MT aus
"MX_MT_Reset_Anf"	M 241.4	BOOL	// MESSTASTER: Reset Taster Anforderung
"MX_Prog_Ende_Flanke"	M 241.5	BOOL	// MA: Programm Ende Flanke positiv
"MX_MT_Flanke_WZW"	M 241.6	BOOL	// MESSTASTER: Flanke WZW
"M_SOKO_NC_STARTSPERRE"	M 241.7	BOOL	// SONDERKONSTRUKTION: NC-Startsperre von SOKO
"M_7Achse_existiert"	M 244.0	BOOL	// AX: 7-Achse ist existent
"M_8Achse_existiert"	M 244.1	BOOL	// AX: 8-Achse ist existent
"M_9Achse_existiert"	M 244.2	BOOL	// AX: 9-Achse ist existent
"M_SPF_eingeschaltet"	M 244.3	BOOL	// SPF: Spaenefoerderer in Betrieb
"M_8Achse_Cam_Aktiv"	M 244.4	BOOL	// AX: 8-Achse Softwarenocken aktiv
"M_15Achse_Cam_Aktiv"	M 244.5	BOOL	// AX: 15-Achse Softwarenocken aktiv
"M_11Achse_existiert"	M 244.6	BOOL	// AX: 11-Achse ist existent
"M_12Achse_existiert"	M 244.7	BOOL	// AX: 12-Achse ist existent
"M_MZU_M_Ready_Flanke_pos"	M 245.0	BOOL	// MZU: Ready M-Funktion Flanke positiv
"M_Ausg_M180_aktiv"	M 245.1	BOOL	// M-AUSGANG: MZU: Merker Ausgaenge M180 aktiv
"M_Ausg_M181_aktiv"	M 245.2	BOOL	// M-AUSGANG: MZU: Merker Ausgaenge M181 aktiv
"M_Ausg_M182_aktiv"	M 245.3	BOOL	// M-AUSGANG: MZU: Merker Ausgaenge M182 aktiv
"M_Ausg_M183_aktiv"	M 245.4	BOOL	// M-AUSGANG: MZU: Merker Ausgaenge M183 aktiv
"M_Ausg_M184_aktiv"	M 245.5	BOOL	// M-AUSGANG: MZU: Merker Ausgaenge M184 aktiv
"M_Ausg_M185_aktiv"	M 245.6	BOOL	// M-AUSGANG: MZU: Merker Ausgaenge M185 aktiv
"M_Ausg_M186_aktiv"	M 245.7	BOOL	// M-AUSGANG: MZU: Merker Ausgaenge M186 aktiv
"M_Ausg_M187_aktiv"	M 246.0	BOOL	// M-AUSGANG: MZU: Merker Ausgaenge M187 aktiv
"M_Ausg_M188_aktiv"	M 246.1	BOOL	// M-AUSGANG: MZU: Merker Ausgaenge M188 aktiv
"M_Ausg_M189_aktiv"	M 246.2	BOOL	// M-AUSGANG: MZU: Merker Ausgaenge M189 aktiv
"M_M161_aktiviert"	M 246.3	BOOL	// KM: M161 (Spänespülung) angewählt
"M_M162_aktiviert"	M 246.4	BOOL	// KM: M162 (Werkstückspülung) angewählt
"M_4Achse_Cam_Aktiv"	M 246.5	BOOL	// AX: 4-Achse Softwarenocken aktiv
"M_5Achse_Cam_Aktiv"	M 246.6	BOOL	// AX: 5-Achse Softwarenocken aktiv
"M_4Achse_existiert"	M 248.0	BOOL	// AX: 4-Achse ist existent
"M_5Achse_existiert"	M 248.1	BOOL	// AX: 5-Achse ist existent
"M_6Achse_existiert"	M 248.2	BOOL	// AX: 6-Achse ist existent
"M_RundAchse_aktiv"	M 248.3	BOOL	// AX: Achse aktiv Bit
"M_Achse4_geloest"	M 248.4	BOOL	// AX: Achse 4 wurde geloest
"M_Achse5_geloest"	M 248.5	BOOL	// AX: Achse 5/11 wurde geloest
"M_Achse6_geloest"	M 248.6	BOOL	// AX: Achse 6 wurde geloest
"M_Achse4_loesen"	M 248.7	BOOL	// AX: Achse 4 loesen
"M_Achse5_loesen"	M 249.0	BOOL	// AX: Achse 5/11 loesen
"M_Achse6_loesen"	M 249.1	BOOL	// AX: Achse 6 loesen
"M_Achse4_klemmen"	M 249.2	BOOL	// AX: Achse 4 klemmen
"M_Achse5_klemmen"	M 249.3	BOOL	// AX: Achse 5/11 klemmen
"M_Achse6_klemmen"	M 249.4	BOOL	// AX: Achse 6 klemmen
"M_Achse4_Ready"	M 249.5	BOOL	// AX: Achse 4 Ready mit klemmen/loesen
"M_Achse5_Ready"	M 249.6	BOOL	// AX: Achse 5/11 Ready mit klemmen/loesen
"M_Achse6_Ready"	M 249.7	BOOL	// AX: Achse 6 Ready mit klemmen/loesen
"I_FMS_NC_START"	M 251.2	BOOL	// M-EINGANG: Handlingsystem Start
"M_KMTL_SPALTSIEB_AKTIV"	M 252.0	BOOL	// KM: Spaltsieb Reinigungsablauf aktivieren
"M_KMTL_SPALTSIEB_GEREINI"	M 252.1	BOOL	// KM: Spaltsieb gereinigt
"M_10Achse_existiert"	M 253.0	BOOL	// AX: 10-Achse ist existent
"M_A5_loes_aktiv"	M 253.1	BOOL	// AX: Achse 5/11  loesen ist aktiv
"M_16Achse_existiert"	M 253.2	BOOL	// AX: 16-Achse ist existent
"M_Tr_pos_Ax4"	M 253.4	BOOL	// AX: Fahranforderung Achse 4 Flanke positiv
"M_Tr_pos_Ax5"	M 253.5	BOOL	// AX: Fahranforderung Achse 5/11 Flanke positiv
"Mx_TPF_Motor_ein"	M 253.6	BOOL	// KM: Motor ein Papierbandfilter
"M_Tr_neg_Ax4"	M 253.7	BOOL	// AX: Fahranforderung Achse 4 Flanke negativ
"M_Tr_neg_Ax5"	M 254.0	BOOL	// AX: Fahranforderung Achse 5/11 Flanke negativ
"I_FMS_APC_MOVEMENT_OK"	M 254.1	BOOL	// M-EINGANG: Handlingsystem APC movement ok
"mx_kanal1_h2_change"	M 254.3	BOOL	// H function 2 Change
"mx_kanal1_h3_change"	M 254.4	BOOL	// H function 3 Change
"MX_AX4_O_Klemm_Auf"	M 254.5	BOOL	// AX: Achse 4 Temporärer Ausgang Klemmung Auf
"MX_AX5_O_Klemm_Auf"	M 254.6	BOOL	// AX: Achse 5/11 Temporärer Ausgang Klemmung Auf
"MX_AX4_Klemm_Aktiv"	M 254.7	BOOL	// AX: Achse 4 Klemmvorgang Aktiv
"MX_AX4_FP1_FUe"	M 255.1	BOOL	// AX: Achse 4 Flanke Fehlerüberwachung
"MX_AX4_FP2_FUe"	M 255.2	BOOL	// AX: Achse 4 Flanke Fehlerüberwachung
"MX_AX5_FP1_FUe"	M 255.3	BOOL	// AX: Achse 5/11 Flanke Fehlerüberwachung
"MX_AX5_FP2_FUe"	M 255.4	BOOL	// AX: Achse 5/11 Flanke Fehlerüberwachung
"MX_Pal_auf_Stoerung"	M 255.5	BOOL	// RS4: Palette wurde auf Störung gesetzt (WZ-Bruch)
"M_FP_IKZ_Taste"	M 260.0	BOOL	// KM: Taste Innere Kühlmittelzufuhr Flanke positiv
"M_FP_KMTL_Taste"	M 260.1	BOOL	// KM: Taste Kühlmittel Flanke positiv
"M_IKZ_Taste"	M 260.2	BOOL	// KM: Taste Innere Kühlmittelzufuhr
"M_KMTL_Taste"	M 260.3	BOOL	// KM: Taste Kühlmittel
"M_M7_Act"	M 260.4	BOOL	// KM: M7 Aktiv
"M_M8_Act"	M 260.5	BOOL	// KM: M8 Aktiv
"M_Fehler_Kmtl_Anlage"	M 260.6	BOOL	// KM: Fehler in Kühlmittelanlage
"M_Umschalt_KMTL"	M 260.7	BOOL	// KM: Umschaltung Wasser/Luft  1=Luft
"M_FP_T_SPL_AKTIV"	M 261.0	BOOL	// FRÄS-DREHTISCH SCHMIERUNG: Zyklenschalter Progressivverteiler
"M_FP_T_FD_SCHMIER_WAR"	M 261.1	BOOL	// FRÄS-DREHTISCH SCHMIERUNG: Warnung Flanke positiv
"M_HR_bereit"	M 261.2	BOOL	// MSST: Handrad bereit
"M_FP_O_FDSchmierung"	M 261.3	BOOL	// FRÄS-DREHTISCH SCHMIERUNG: Einschalten Flanke positiv
"mx_kanal_1_h1_change"	M 261.4	BOOL	// H function 1 Change
"M_FN_T_FD_SCHMIER_WAR"	M 261.5	BOOL	// FRÄS-DREHTISCH SCHMIERUNG: Warnung Flanke negativ
"M_M8_WZ_Tab"	M 261.6	BOOL	// KM: Anwahl Kühlmittel 1 in WZ-Liste
"M_M7_WZ_Tab"	M 261.7	BOOL	// KM: Anwahl Kühlmittel 2 in WZ-Liste
"MX_FP_EinwRdy"	M 268.0	BOOL	// WZW: Werkzeug eingewechselt Flanke positiv
"I_WZB_Parkstellung"	M 268.1	BOOL	// M-EINGANG: Bruchüberwachung in Parkstellung
"M_Umsp_Gr1_WZListe"	M 268.2	BOOL	// WZV: Umspeichern Greifer 1 in Werkzeugliste
"M_Umsp_Gr2_WZListe"	M 268.3	BOOL	// WZV: Umspeichern Greifer 2 in Werkzeugliste
"M_Umsp_WZListe_Gr2"	M 268.4	BOOL	// WZV: Umspeichern Werkzeugliste in Greifer 2
"M_WZV_Regal_Done"	M 268.5	BOOL	// WZV OMRON: Done
"M_WZV_Regal_Error"	M 268.6	BOOL	// WZV OMRON: Error
"M_IM_Taste_Tuerver_entr"	M 268.7	BOOL	// MA: Impuls Kabinentür entriegeln
"M_A6_loes_aktiv"	M 269.0	BOOL	// AX: Achse 6 Klemmung lösen aktiv
"M_Tr_pos_Ax6"	M 269.1	BOOL	// AX: Fahranforderung Achse 6 Flanke positiv
"M_Tr_neg_Ax6"	M 269.2	BOOL	// AX: Fahranforderung Achse 6 Flanke negativ
"MX_AX6_O_Klemm_Auf"	M 269.3	BOOL	// AX: Achse 6 Temporärer Ausgang Klemmung Auf
"MX_AX6_FP1_FUe"	M 269.4	BOOL	// AX: Achse 6 Flanke Fehlerüberwachung
"MX_AX6_FP2_FUe"	M 269.5	BOOL	// AX: Achse 6 Flanke Fehlerüberwachung
"M_RF_6ACHS"	M 269.6	BOOL	// AX: Achse 6 XXX
"M_FN_3te_BA"	M 270.0	BOOL	// MA: 4 Betriebsart Flanke negativ
"M_FP_Luftkuehlung"	M 270.1	BOOL	// Schmierung Drehdurchführung Luftkühlung ein Flanke positiv
"M_Imp_Luftkuehlung_ein"	M 270.2	BOOL	// Schmierung Drehdurchführung Luftkühlung ein Impuls
"HM_PI_Takt_02s"	M 270.3	BOOL	// Takt 0.2sec Flanke positiv
"M_FP_Takt_02s"	M 270.4	BOOL	// Takt 0.2sec Impuls
"I_KM_FILTER_FEINB_OK"	M 270.5	BOOL	// ME B3-90.3 Filter Feinst-Bereich OK
"Mx_FP_Taste_WZ_Achse_RET"	M 270.7	BOOL	// Werkzeugachse Rettung Impuls positiv
"M_BR_CAX_ZU_ZD"	M 280.0	BOOL	// AX: Achse 4 Bei ZD Bremse C-Achse Schliessen
"M_TPrepare_Quit"	M 280.1	BOOL	// WZV: Werkzeug vorbereiten Quittierung
"I_WW_NEG_MSS"	M 280.2	BOOL	// M-EINGANG: Motorschutzschalter Werkzeugwechsler
"I_AL_TASTER_WZ_SPA"	M 280.4	BOOL	// M-EINGANG: Taster Werkzeugspanner geloest
"I_FD_KA_Fuellstand"	M 281.0	BOOL	// M-EINGANG: Kuehlaggregat Fraes-Drehtisch Fuellstand
"I_FD_KA_NEG_Durchflussw"	M 281.1	BOOL	// M-EINGANG: Kuehlaggregat Fraes-Drehtisch Durchflusswaechter
"I_FD_KA_NEG_Luftfilter"	M 281.2	BOOL	// M-EINGANG: Kuehlaggregat Fraes-Drehtisch Filterverschmutzung
"I_FD_KA_NEG_Sammelfehler"	M 281.3	BOOL	// M-EINGANG: Motorschutzschalter Spindelkuehlung
"I_FD_KA_Temperaturregler"	M 281.4	BOOL	// M-EINGANG: Kuehlaggregat Fraes-Drehtisch Temperaturregler
"I_FD_Tisch_geklemmt"	M 281.5	BOOL	// M-EINGANG: Klemmung Fraes-Drehtisch geklemmt
"I_FD_Tisch_geloest_1"	M 281.6	BOOL	// M-EINGANG: Klemmung Fraes-Drehtisch geloest
"I_FD_TISCHTEMP_NOTAUS"	M 281.7	BOOL	// M-EINGANG: Temperaturueberwachung Motor Fraes-Drehtisch
"I_KM_DRUCK2_M7_ENABLE"	M 282.0	BOOL	// M-EINGANG: Kuehlmittel Filterverschmutzung Feinstbereich
"I_SPI_geklemmt"	M 282.1	BOOL	// M-EINGANG: Ueberwachung Fraesspindel geklemmt
"I_SPI_geloest"	M 282.2	BOOL	// M-EINGANG: Ueberwachung Fraesspindel geloest
"I_TA_KLEMMUNG_GELOEST"	M 282.3	BOOL	// M-EINGANG: Klemmung geloest NC-Teilapparat
"m_282.4"	M 282.4	BOOL	// Reserve
"O_FD_BETRIEBSTUNDE"	M 282.5	BOOL	// M-AUSGANG: Fraes-Drehtisch Betriebsstundenzaehler
"O_FD_Tisch_klemmen"	M 282.6	BOOL	// M-AUSGANG: Klemmung Fraes-Drehtisch klemmen
"O_FD_Tisch_loesen"	M 282.7	BOOL	// M-AUSGANG: Klemmung Fraes-Drehtisch loesen
"O_KM_DRUCK2_M7_EIN"	M 283.0	BOOL	// M-AUSGANG: Hochdruckpumpe Kuehlmittel 2 80 bar
"O_SPI_klemmen"	M 283.1	BOOL	// M-AUSGANG: Fraesspindel klemmen
"O_SPI_loesen"	M 283.2	BOOL	// M-AUSGANG: Fraesspindel loesen
"O_KM_DRUCK2_M7_VORHANDEN"	M 283.3	BOOL	// M-AUSGANG: Hochdruckpumpe Kuehlmittel 2 80 bar vorhanden
"m283.4"	M 283.4	BOOL	// Reserve
"Mx_Freigabe_DS"	M 283.5	BOOL	// KM: Freigabe Druckstufen
"M_Reset_Druckstufen"	M 283.6	BOOL	// KM: Reset Druckstufen
"MX_DS1_AKtiv"	M 283.7	BOOL	// KM: Druckstufe 1 aktiv
"MX_ASpdl_M3_Aktiv"	M 284.0	BOOL	// AX4: (C-Achse) M3 (Rechtslauf) aktiv
"MX_ASpdl_M4_Aktiv"	M 284.1	BOOL	// AX4: (C-Achse) M3 (Linksslauf) aktiv
"MX_ASpdl_FP_M4"	M 284.2	BOOL	// AX4: (C-Achse) M4 (Linksslauf) aktiv Flanke positiv
"MX_ASpdl_FP_M3"	M 284.3	BOOL	// AX4: (C-Achse) M3 (Rechtslauf) aktiv Flanke positiv
"MX_ASpdl_FP_M5"	M 284.4	BOOL	// AX4: (C-Achse) M5 (Aus) aktiv Flanke positiv
"MX_DS2_Aktiv"	M 284.5	BOOL	// KM: Druckstufe 2 aktiv
"MX_DS3_Aktiv"	M 284.6	BOOL	// KM: Druckstufe 3 aktiv
"MX_DS4_Aktiv"	M 284.7	BOOL	// KM: Druckstufe 4 aktiv
"MX_DS5_Aktiv"	M 285.0	BOOL	// KM: Druckstufe 5 aktiv
"MX_DS6_Aktiv"	M 285.1	BOOL	// KM: Druckstufe 6 aktiv
"Mx_DX7_aktiv"	M 285.2	BOOL	// KM: Druckstufe 7 aktiv
"MX_IKZ_Freigabe_Vorschub"	M 285.3	BOOL	// KM: Vorschubfreigabe von innerer Kühlmittelzufuhr
"M_FP_H30"	M 285.4	BOOL	// KM: H-Funktion 7 Flanke positiv
"O_KM_DRUCK3_M7_EIN"	M 285.5	BOOL	// AUSGANG: KM Druck 3 M7 ein
"MX_IKZ_Pumpen_Ein"	M 285.6	BOOL	// KM: Pumpen für innere Kühlmittelzufuhr einschalten
"I_KM_DRUCK1_M7_ENABLE"	M 285.7	BOOL	// M-EINGANG: KM Druck 1 M7 Freigabe
"I_KM_SPRUEHPIST_RPL_EIN"	M 286.0	BOOL	// M-EINGANG: Anforderung Spülpistole Rüstplatz Ein
"I_Stern_4Ax"	M 286.1	BOOL	// M-EINGANG:
"O_KM_SPRUEHPIST_RPL_EIN"	M 286.2	BOOL	// M-AUSGANG: Signalleuchte Spülpistole Rüstplatz Ein
"O_Stern_4Ax"	M 286.3	BOOL	// M-AUSGANG:
"I_KM_DRUCK1_M7_EIN"	M 286.4	BOOL	// M-EINGANG:
"O_KM_DRUCK1_M7_EIN"	M 286.5	BOOL	// AUSGANG: KM Druck 1 M7 ein
"MX_Freigabe_KM_30Bar"	M 286.6	BOOL	// Freigabe von M7 bis 30 Bar bei U-Achse
"MX_FREIG_ANAL_80BAR"	M 286.7	BOOL	// Freigabe analoge Druckstufe  mit einem Proportionalventil 0-80 Bar
"M_WK_GRF_AST_1"	M 287.0	BOOL	// Winkelkopfwechsler: Motor Greiferarm in Arbeitsstellung 1
"M_WK_GRF_AST_2"	M 287.1	BOOL	// Winkelkopfwechsler: Motor Greiferarm in Arbeitsstellung 2
"M_WK_GRF_GST"	M 287.2	BOOL	// Winkelkopfwechsler: Motor Greiferarm in Grundstellung
"M_FP_WFK_GRF_Z_VOR"	M 287.3	BOOL	// Flankenmerker: Winkelkopfwechsler Motor Vorwärts
"M_FP_WFK_GRF_Z_RUECK"	M 287.4	BOOL	// Flankenmerker: Winkelkopfwechsler Motor Rückwärts
"Mx_Werkzeugdaten_lesen"	M 288.0	BOOL	// WZV: Request Greiferdaten lesen
"Mx_WZdaten_lesen_ready"	M 288.1	BOOL	// WZV: Greiferdaten lesen fertig
"M_WZDaten_lesen_ready_S"	M 288.2	BOOL	// WZV: Greiferdaten lesen fertig (gespeichert)
"Mx_Wzdaten_lesen_error"	M 288.3	BOOL	// WZV: Error Greiferdaten lesen
"HM_PI_WZD_lesen_ready"	M 288.6	BOOL	// WZV: Greiferdaten lesen fertig Flanke positiv
"O_MinSchm_IKZ_ausblasen"	M 288.7	BOOL	// KM: Minimalmengen Schmierung: Leitung bei M7 ausblasen
"M_WZV_Bereitst_Fertig"	M 290.0	BOOL	// WZV: Quittung Bereitstellen fertig
"M_WZV_Spi_Mag"	M 290.1	BOOL	// WZV: Umspeichern Spindel nach Magazin
"M_WZV_Mag_Spi"	M 290.2	BOOL	// WZV: Umspeichern Magazin nach Spindel
"M_WZV_Gr2_Mag"	M 290.3	BOOL	// WZV: Umspeichern Greifer 2 nach Magazin
"M_WZV_Beladen_ende"	M 290.4	BOOL	// WZV: Beladen beendet
"M_WZV_Entladen_ende"	M 290.5	BOOL	// WZV: Entladen beendet
"M_WZV_Entladen_Abbruch"	M 290.6	BOOL	// WZV: Be/Entladen abgebrochen
"M_WZV_Vorber_Req"	M 291.0	BOOL	// WZV: Anforderung WZ bereitstellen
"Mx_WZ_Ablegen_Rettung"	M 291.1	BOOL	// WZV: Werkzeug ablegen aus Rettung
"M_WZV_Positionieren"	M 291.3	BOOL	// WZV: Positionieren beendet
"I_WM_WZ_einlegen"	M 291.4	BOOL	// M-EINGANG: Quittierung Werkzeug einlegen
"I_WM_WZ_entnehmen"	M 291.5	BOOL	// M-EINGANG: Quittierung Werkzeug entnehmen
"M_WZV_Gr1_Mag"	M 291.6	BOOL	// WZV: Umspeichern Greifer 1 nach Magazin
"M_WZV_Quit_Bereitst"	M 291.7	BOOL	// WZV: Quittierung Bereitstellen fertig
"M_Umsp_Gr1-Mag"	M 295.1	BOOL	// WZW: Umspeichern Greifer 1 zu Magazin
"M_Umsp_Gr2-Spdl"	M 295.2	BOOL	// WZW: Umspeichern Greifer 2 zu Spindel
"M_WZ_Reinigen"	M 295.3	BOOL	// WZW: Anforderung WZ Vorbereiten
"M_WZ_Reinigen_RDY"	M 295.4	BOOL	// WZW: Rueckmeldung WZ Vorbereiten
"M_Req_Ablegen_WZ"	M 295.5	BOOL	// WZW: Anforderung WZ Ablegen
"M_Req_WZ_Reinigen"	M 295.7	BOOL	// WZW: Anforderung Reinigen WZ
"M_Ready_WZ_Reinigen"	M 296.0	BOOL	// WZW: Rueckmmeldung WZ Reinigung
"M_WZKR_Beweg"	M 296.2	BOOL	// WZW: Kegelreinigung in Bewegung
"M_WZR_Mag_Verrieg"	M 296.3	BOOL	// WZW: Verriegelung Magazin
"M_WZ_Rdy_Ablegen"	M 296.4	BOOL	// WZW: Ablegen Werkzeug
"M_WZ_Reinigen_Aktiv"	M 296.6	BOOL	// WZW: Vorbereiten aktiv
"M_WiKo_Wechsel_aktiv"	M 297.1	BOOL	// WIKO: Wechsel Wiegenfräskopf aktiv
"M_Frg_Hub_MagPos"	M 297.2	BOOL	// Freigabe Hub Richtung Magazinposition
"M_Magazin_Sperre"	M 297.3	BOOL	// MAG: Sperre Magazin
"M_MA_Fehler_ER_Modul"	M 297.4	BOOL	// MA: Fehler ER Modul
"M_MA_Entprell_ER"	M 297.5	BOOL	// MA: Entprellbit Überwachung ER Modul
"M_MA_Hydr_Perm_Pumpen"	M 297.6	BOOL	// MA: Ansteuerung Hydraulik permanent pumpen
"M_Jog_Req_4Ax_Plus_Minus"	M 297.7	BOOL	// AX: 4.Achse Plus/Minus Jog-Fahranforderung
"M_req_WZ_entriegeln"	M 298.0	BOOL	// WZW: Anforderung Werkzeug entriegeln im Magazin
"M_req_WZ_verriegeln"	M 298.1	BOOL	// WZW: Anforderung Werkzeug verriegeln im Magazin
"M_req_Greifer_ausfahren"	M 298.2	BOOL	// WZW: Anforderung Greifer ausfahren
"M_req_Greifer_einfahren"	M 298.3	BOOL	// WZW: Anforderung Greifer einfahren
"MX_Jobbearbeitung"	M 298.6	BOOL	// STA: Maschine in Jobbearbeitung
"M_Frg_Hub_SpiPos"	M 298.7	BOOL	// Freigabe Hub Richtung Spindelposition
"I_WW_GRF_ENTRIEGELT"	M 299.0	BOOL	// M-EINGANG: Verriegelung Werkzeuggreifer entriegelt
"O_WW_GRF_ENTRIEGELN"	M 299.1	BOOL	// M-AUSGANG: Verriegelung Werkzeuggreifer entriegeln
"m_299.2"	M 299.2	BOOL	// Reserve
"MX_FP_YD_Schalten"	M 299.3	BOOL	// SternDr: Flanke YD geschaltet
"M_Umsp_Spdl_Gr1"	M 299.4	BOOL	// WZW: BefA umspeichern Spindel zu Greifer 1
"M_neue_Pal_anwaehlen"	M 299.5	BOOL	// PRG: Neue Palette anwählen
"M_EINL_SP_B_UNTERBRECHEN"	M 299.6	BOOL	// Unterbrechung Einlesesperre Takttisch gelöst bei WZW
"m_299.7"	M 299.7	BOOL	// Reserve
"m_300.0"	M 300.0	BOOL	// Reserve
"m_300.1"	M 300.1	BOOL	// Reserve
"Mx_X_ACHSE_WZW_POS"	M 300.2	BOOL	// WZW: X-Achse auf Wechselpos, X-Achse ausserhalb von WZW-Klappe
"m_300.3"	M 300.3	BOOL	// Reserve
"m_300.4"	M 300.4	BOOL	// Reserve
"m_300.5"	M 300.5	BOOL	// Reserve
"m_300.6"	M 300.6	BOOL	// Reserve
"m_300.7"	M 300.7	BOOL	// Reserve
"mx_fn_achs5"	M 301.0	BOOL	// AX: Achse 5 Reglerfreigabe
"m_301.1"	M 301.1	BOOL	// Reserve
"m_301.4"	M 301.4	BOOL	// Reserve
"m_301.5"	M 301.5	BOOL	// Reserve
"m_301.6"	M 301.6	BOOL	// Reserve
"I_DM_Ta_SKR_gelb"	M 301.7	BOOL	// RS4: MSST: Taste Bild links gelb
"I_DM_Ta_SKR_blau"	M 302.0	BOOL	// RS4: MSST: Taste Bild rechts lila
"m_302.1"	M 302.1	BOOL	// Reserve
"m_302.3"	M 302.3	BOOL	// Reserve
"m_302.5"	M 302.5	BOOL	// Reserve
"I_PW_HUB_POSITION_4"	M 302.7	BOOL	// M-EINGANG: Palettenwechsler Hub Position 4
"MX_Rundspeicher_RS4"	M 303.0	BOOL	// PALETTENSPEICHER: Rundspeicher RS4 angewaehlt
"m_PW_Abbruch_Fastems"	M 303.1	BOOL	// Abbruch Palettenwechsler bei Betrieb mit Fastems
"M_Grf2_entr_req"	M 304.0	BOOL	// WZV: Anforderung Greifer 2 entriegeln
"M_Grf2_verr_req"	M 304.1	BOOL	// WZV: Anforderung Greifer 2 verriegeln
"m_305.7"	M 305.7	BOOL	// RS4: Anforderung Palette von Maschine holen
"M_JOPBETRIEB_FP"	M 306.0	BOOL	// RS4: Jobbetrieb Flanke positiv
"MX_Kein_JOB_Vorhanden"	M 306.1	BOOL	// PRG: Kein Job vorhanden
"MX_Job_In_Maschine"	M 306.2	BOOL	// PRG: Job in Maschine
"MX_Job_RP"	M 306.3	BOOL	// PRG: Job auf Rüstplatz
"MX_Jobbetrieb"	M 306.4	BOOL	// PRG: Jobbetrieb
"Mx_Verlasse_Prg"	M 306.5	BOOL	// PRG: Programm verlassen
"MX_Prg_von_Maschine"	M 306.6	BOOL	// PRG: Programm von Maschine angewaehlt
"M_Prg_Maschine_anwaehl"	M 306.7	BOOL	// PRG: Maschine anwählen
"I_WZ-Spanner_Gesp_mit_WZ"	M 307.0	BOOL
"M_FP_Prg_Masch_gestartet"	M 307.1	BOOL	// PRG: Programm von Maschine gestartet Flanke positiv
"M_PWMakro_NCStart"	M 307.3	BOOL	// PRG: Paletenwechsler Makro NC-Start
"M_FP_NCStart_RS4_PW"	M 307.4	BOOL	// PRG: Paletenwechsler Makro NC-Start Flanke positiv
"I_D_PW_HUB_POS2"	M 307.7	BOOL	// M-EINGANG: Palettenwechsler Diagnose Position 2
"M_Request_TDS"	M 308.0	BOOL	// TDS: BALLUFF Anstoss FC197 aus FC193
"M_TDS_WZ_NC_DELET"	M 308.1	BOOL	// TDS: BALLUFF Werkzeug NC löschen
"M_FP_Request"	M 308.2	BOOL	// TDS: BALLUFF Anstoss FC197 aus FC193 Flanke positiv
"M_Request_TDS_bel"	M 308.3	BOOL	// TDS: BALLUFF Start beladen
"M_FP_Request_bel"	M 308.4	BOOL	// TDS: BALLUFF Start beladen Flanke positiv
"M_TDS_RUNS"	M 308.5	BOOL	// TDS: BALLUFF TDS läuft
"M_ENTLADEN_TDS"	M 308.6	BOOL	// TDS: BALLUFF Konfiguration WZ entladen über TDS
"M_ANF_TNR_LESEN"	M 309.0	BOOL	// TDS: BALLUFF WZ-Nummer aus WZ-Listen über FB228 lesen
"M_Request_FB228"	M 309.1	BOOL	// TDS: BALLUFF WZ-Nummer aus WZ-Listen lesen gespeichert
"M_DONE_FB228"	M 309.2	BOOL	// TDS: BALLUFF WZ-Nummer aus WZ-Listen gelesen
"M_DONE_TNR_LESEN"	M 309.3	BOOL	// TDS: BALLUFF WZ-Nummer aus WZ-Listen gelesen gespeichert
"M_FP_ANF_FB228"	M 309.4	BOOL	// TDS: BALLUFF WZ-Nummer aus WZ-Listen lesen Flanke positiv
"M_NC_lesen_beladen"	M 309.5	BOOL	// TDS: BALLUFF WZ-Nummer gelesen beim Beladen
"M_Error_Beladen"	M 309.6	BOOL	// TDS: BALLUFF Fehler beim beladen falsches WZ beim lesen
"I_PW_RPL_FREIGABE"	M 309.7	BOOL	// M-EINGANG: Antriebsfreigabe Ruestplatz
"MX_RS_HUB_BEWEGUNG"	M 310.0	BOOL	// PALETTENSPEICHER: Hub Bewegung aktiv
"M_NCSNR_lesen"	M 310.1	BOOL	// WIKO: Neuen Schritt von NC lesen
"MX_RS_KLM_BEWEGUNG"	M 310.2	BOOL	// PALETTENSPEICHER: KLM Bewegung
"I_PW_RPL_links_drehen"	M 310.3	BOOL	// M-EINGANG: Ruestplatz drehen Links
"I_PW_RPL_rechts_drehen"	M 310.4	BOOL	// M-EINGANG: Ruestplatz drehen Rechts
"I_PW_RPL_ZUSTIMMTASTE"	M 310.5	BOOL	// M-EINGANG: Zustimmungstaste NC-Ruestplatz drehen
"O_PW_RPL_BREMSE_AUF"	M 310.6	BOOL	// M-AUSGANG: Bremse NC-Ruestplatz Auf
"O_PW_RPL_FREIGABE_RE_LI"	M 310.7	BOOL	// M-AUSGANG: Freigabe NC-Ruestplatz
"M_LS_Fehl"	M 315.0	BOOL	// PALETTENSPEICHER: Fehler
"M_LS_Ax_10_11_Freig"	M 315.1	BOOL	// PALETTENSPEICHER: Leistung für RS-Achsen zuschalten
"M_LS_FP_SKR"	M 315.2	BOOL	// PALETTENSPEICHER: OEM Einrichten aktiv Flanke positiv
"MX_POS_FL_SKR"	M 315.3	BOOL	// PALETTENSPEICHER: OEM Einrichten aktiv Impuls
"MX_Transport_Gst"	M 315.4	BOOL	// PALETTENSPEICHER: Transport in Grundstellung
"M_RS_RETTUNG_AKTIV"	M 315.5	BOOL	// PALETTENSPEICHER: Rettung aktiv
"M_DS_Pos_2"	M 315.6	BOOL	// PALETTENSPEICHER: Drehstation Position Rüstplatz
"M_DS_Pos_3"	M 315.7	BOOL	// PALETTENSPEICHER: Drehstation  Position Übergabeplatz
"M_DS_Pos_4"	M 316.0	BOOL	// PALETTENSPEICHER: Drehstation Position Speicherplatz 1
"M_DS_Pos_5"	M 316.1	BOOL	// PALETTENSPEICHER: Drehstation Position Speicherplatz 2
"M_DS_Pos_6"	M 316.2	BOOL	// PALETTENSPEICHER: Drehstation Position Speicherplatz 3
"MX_Transport_Ausgef"	M 316.3	BOOL	// PALETTENSPEICHER: Transport ausgefahren
"MX_RS_Grundstellung"	M 316.4	BOOL	// PALETTENSPEICHER: In Grundstellung
"MX_UG_Auftrag"	M 316.5	BOOL	// PALETTENSPEICHER: Maschinenübergabeauftrag
"MX_RPL_Auftrag"	M 316.6	BOOL	// PALETTENSPEICHER: Rüstplatzauftrag
"M_DS_Pos_7"	M 316.7	BOOL	// PALETTENSPEICHER: Drehstation Position Speicherplatz 4
"M_FRG_Drehst_Achse"	M 317.0	BOOL	// PALETTENSPEICHER: Freigabe Drehstation Achse
"M_FRG_Transp_Achse"	M 317.1	BOOL	// PALETTENSPEICHER: Freigabe Transport Achse
"M_FN_Speicher"	M 317.2	BOOL	// PALETTENSPEICHER: Leistung für RS-Achse zuschalten Flanke negativ
"M_RS4_80er"	M 317.3	BOOL	// PALETTENSPEICHER: RS4 80er aktiv
"M_FRG_Hub_Achse"	M 317.4	BOOL	// PALETTENSPEICHER: Freigabe Hub-Achse
"MX_ABST_Rundspeicher"	M 317.5	BOOL	// PALETTENSPEICHER: Ausbaustufe: Rundspeicher aktiv
"HM_NI_Bew_39_211"	M 317.6	BOOL	// PALETTENSPEICHER: Bewegung 39 oder 211 Plus oder Minus Flanke negativ
"MX_RS_HUB_Fertig"	M 317.7	BOOL	// PALETTENSPEICHER: Hubachse Position erreicht
"M_RS_HUBACHSE_BER_EBENE0"	M 318.0	BOOL	// PALETTENSPEICHER: Hubachse im Bereich Ebene 0
"M_RS_HUBACHSE_BER_EBENE1"	M 318.1	BOOL	// PALETTENSPEICHER: Hubachse im Bereich Ebene 1
"MX_SKR_HUB_Req"	M 318.2	BOOL	// PALETTENSPEICHER: Hub-Achse Fahranforderung
"MX_RS_DrehSt_Fertig"	M 318.3	BOOL	// PALETTENSPEICHER: Drehstation Position erreicht
"MX_RS_Tansport_Fertig"	M 318.4	BOOL	// PALETTENSPEICHER: Transport Position erreicht
"M_RS_SKR_NEG"	M 318.5	BOOL	// PALETTENSPEICHER: RS OEM Einrichten aktiv Flanke negativ
"MX_SKR_FP_RS"	M 318.6	BOOL	// PALETTENSPEICHER: RS OEM Einrichten aktiv Flanke positiv
"eax_9.AX_Bremse_oeffnen"	M 318.7	BOOL	// AX: Achse 9 Bremse lüften
"m_PS_STOP_TUERE_NICHT_ZU"	M 319.0	BOOL	// PS: Transport PS gestoppt, tueren nicht zu
"MX_SKR_DSt_Req"	M 319.1	BOOL	// PALETTENSPEICHER: Drehstation Fahranforderung
"MX_SKR_Trp_Req"	M 319.2	BOOL	// PALETTENSPEICHER: Transport Fahranforderung
"M_RS_FP_Oem4"	M 319.3	BOOL	// PALETTENSPEICHER: Bewegung 35 Plus oder Minus Flanke negativ
"M_RS_FP_Oem2"	M 319.4	BOOL	// PALETTENSPEICHER: Bewegung 32 bis 34 Plus oder Minus Flanke negativ
"M_RS_FN_Oem3"	M 319.5	BOOL	// PALETTENSPEICHER: Leistung für Rundspeicherachse Flanke negativ 1
"M_RS_FN_Oem5"	M 319.6	BOOL	// PALETTENSPEICHER: Leistung für Rundspeicherachse Flanke negativ 2
"M_RS_FP_Oem"	M 319.7	BOOL	// PALETTENSPEICHER: Bewegung 36 oder 37 Plus oder Minus Flanke negativ
"M_RS_FP_TRANSPORT"	M 320.0	BOOL	// PALETTENSPEICHER: Transport Maschine zu Speicher Flanke positiv
"M_DS_Pos_8"	M 320.1	BOOL	// PALETTENSPEICHER: Drehstation Position Speicherplatz 5
"M_DS_Pos_9"	M 320.2	BOOL	// PALETTENSPEICHER: Drehstation Position Speicherplatz 6
"M_DS_Pos_10"	M 320.3	BOOL	// PALETTENSPEICHER: Drehstation Position Speicherplatz 7
"M_DS_Pos_11"	M 320.4	BOOL	// PALETTENSPEICHER: Drehstation Position Speicherplatz 8
"M_DS_Pos_12"	M 320.5	BOOL	// PALETTENSPEICHER: Drehstation Position Speicherplatz 9
"M_DS_Pos_13"	M 320.6	BOOL	// PALETTENSPEICHER: Drehstation Position Speicherplatz 10
"M_RS_FN_Oem6"	M 320.7	BOOL	// PALETTENSPEICHER: Leistung für Rundspeicherachse Flanke negativ 3
"M_TM_TPU_GET_TOOL"	M 321.0	BOOL	// WZW: Transporteinheit ist auf Werkzeugkegel gefahren
"M_TM_TPU_RELEASE_TOOL"	M 321.1	BOOL	// WZW: Transporteinheit ist auf Grundstellung gefahren
"M_TM_TPU_TRANSFERPOS"	M 321.2	BOOL	// WZW: Transporteinheit ist zur Übergabeposition gefahren
"M_TM_TPU_MAGAZINPOS"	M 321.3	BOOL	// WZW: Transporteinheit ist zur Magazinpostition gefahren
"M_TM_MAG_TOOL_UNLOCK"	M 321.4	BOOL	// WZW: Werkzeug an Magazinposition ist entriegelt
"M_TM_MAG_TOOL_LOCK"	M 321.5	BOOL	// WZW: Werkzeug an Magazinposition ist verriegelt
"M_TM_TLOAD_TOOL_UNLOCK"	M 321.6	BOOL	// WZW: Werkzeug am Rüstplatz ist entriegelt
"M_TM_TLOAD_TOOL_LOCK"	M 321.7	BOOL	// WZW: Werkzeug am Rüstplatz ist verriegelt
"I_SP_AUFL_ST1_ENTSPANNT"	M 322.0	BOOL	// ME xx-xx.x Kontrolle Auflage Spannstelle 1 entspannt ok
"I_SP_AUFL_ST2_ENTSPANNT"	M 322.1	BOOL	// ME xx-xx.x Kontrolle Auflage Spannstelle 2 entspannt ok
"I_SP_AUFL_ST3_ENTSPANNT"	M 322.2	BOOL	// ME xx-xx.x Kontrolle Auflage Spannstelle 3 entspannt ok
"I_SP_AUFL_ST4_ENTSPANNT"	M 322.3	BOOL	// ME xx-xx.x Kontrolle Auflage Spannstelle 4 entspannt ok
"M_FP_Pal_Störung"	M 322.4	BOOL	// PALETTENSPEICHER: Palette auf Störung setzen Flanke positiv
"M_RS_DREHST_POS_GUELTIG"	M 322.5	BOOL	// PALETTENSPEICHER: Vorgewählte Position Drehstation gültig
"M_RS_DREHST_POSITIONIERT"	M 322.6	BOOL	// PALETTENSPEICHER:  Drehstation positioniert
"M_RS_EINRICHTEN_AKTIV"	M 322.7	BOOL	// PALETTENSPEICHER:  Einrichten aktiv
"M_FP_Umspeichern"	M 324.0	BOOL	// WZV: Umspeichern Flanke positiv
"M_FP_Umspeichern2"	M 324.1	BOOL	// WZV: Umspeichern Flanke positiv 2
"M_FP_Umspeichern3"	M 324.2	BOOL	// WZV: Umspeichern Flanke positiv 3
"M_FP_Umspeichern4"	M 324.3	BOOL	// WZV: Umspeichern Flanke positiv 4
"I_ROBOT_AUTOM_EIN"	M 324.4	BOOL	// ME xx-xx.x Umschaltung Automatikbetrieb Handlingssystem
"O_SP_VORR_ABBLASEN"	M 324.7	BOOL	// MA H4-10.7 Ventil Luft für Vorrichtung Abblasen
"O_AL_LM_RD"	M 327.0	BOOL	// M-AUSGANG: Signalleuchte Farbe RD
"O_AL_LM_YE"	M 327.1	BOOL	// M-AUSGANG: Signalleuchte Farbe YE
"O_AL_LM_GN"	M 327.2	BOOL	// M-AUSGANG: Signalleuchte Farbe GN
"O_AL_LM_BU"	M 327.3	BOOL	// M-AUSGANG: Signalleuchte Farbe BU
"mx_HubUntenNachMitte"	M 327.4	BOOL	// PW: Hub von Unten zur Mitte
"I_KA_NEG_STOERMELDUNG2"	M 327.5	BOOL	// M-EINGANG: Kuehlaggregat Störmeldung Prioritaet 2
"I_KA_NEG_STOERMELDUNG1"	M 327.6	BOOL	// M-EINGANG: Kuehlaggregat Störmeldung Prioritaet 1
"I_KA_NEG_WARNMELDUNG"	M 327.7	BOOL	// M-EINGANG: Kuehlaggregat Warnmeldung
"I_AL_Kabine_zu"	M 332.0	BOOL	// M-EINGANG: Kabinentueren geschlossen
"I_AL_Zustimmtaste"	M 332.1	BOOL	// M-EINGANG: Zustimmungstaste
"I_AL_2_Betriebsart"	M 332.2	BOOL	// M-EINGANG: Betriebsart Einrichten (wird in FC111 negiert)
"I_AL_MASCHINE_EIN"	M 332.3	BOOL	// M-EINGANG: Rueckmeldung Maschine Ein
"I_AL_NEG_SPI_VS_Halt"	M 332.4	BOOL	// M-EINGANG: Spindel/Vorschub Halt
"I_AL_SCH_Rueckmeldung"	M 332.5	BOOL	// M-EINGANG: Druckueberwachung Schmierung Maschine
"I_AL_SCH_Fuellstand"	M 332.6	BOOL	// M-EINGANG: Schmierung Maschine: Fuellstand Schmierstoffpumpe
"I_AL_Tempkomp_TXD"	M 332.7	BOOL	// M-EINGANG: Temperaturkompensation Übernahme Temperaturdaten
"I_AL_1_Stufe_Getriebe"	M 333.0	BOOL	// M-EINGANG: Hauptantrieb 8000 U/min Getriebestellung n<1126 /min
"I_AL_2_Stufe_Getriebe"	M 333.1	BOOL	// M-EINGANG: Hauptantrieb 8000 U/min Getriebestellung n>11126 /min
"I_AL_HYD_Druck_OK"	M 333.2	BOOL	// M-EINGANG: Druckueberwachung Hydraulik
"I_AL_HYD_NEG_Stoerung"	M 333.3	BOOL	// M-EINGANG: Störung Hydraulik (Motorschutzschalter/Temperaturüberwachung)
"I_Taster_WZ_Spanner"	M 333.4	BOOL	// M-EINGANG: Taste Werkzeugspanner gelöst (manuell)
"I_MT_Batterie_low"	M 333.5	BOOL	// M-EINGANG: Messtaster Batteriewarnung
"I_MT_BTB"	M 333.6	BOOL	// M-EINGANG: Messtaster Betriebsbereit
"I_PW_QUIT_Freigabe"	M 333.7	BOOL	// M-EINGANG: Quittierung Freigabe Palettenwechsler
"I_SF_NEG_MSS_Schnecken"	M 334.0	BOOL	// M-EINGANG: Motorschutzschalter Spaenefoerderer Schneckenantrieb
"I_KM_NEG_MSS_SSA"	M 334.1	BOOL	// M-EINGANG: Motorschutzschalter Kuehlmittelanlage
"I_AL_NEG_SAM_ER_Modul"	M 334.2	BOOL	// M-EINGANG: Temperaturüberwachung Versorgungsmodul Antriebe
"I_AL_Kabine_Verriegelt"	M 334.3	BOOL	// M-EINGANG: Kabinentueren verriegelt
"I_HR_Anwahl"	M 334.4	BOOL	// M-EINGANG: Aktivierung Handkommandostation
"I_Ueb_Temp_Sch"	M 334.5	BOOL	// M-EINGANG: Übertemperatur Schaltschrank
"I_SpannDruck_Maschine"	M 334.6	BOOL	// M-EINGANG: Spannvorrichtung Maschine vorhanden
"I_M_T_H_Fkt_fertig"	M 334.7	BOOL	// M-EINGANG: Freigabe T-H- M-Funktionen
"I_SK_HOR_Ebene"	M 335.0	BOOL	// M-EINGANG: Stellung Schwenkfraeskopf waagrecht
"I_SK_VER_Ebene"	M 335.1	BOOL	// M-EINGANG: Stellung Schwenkfraeskopf senkrecht
"I_SK_Klemmung_geklemmt"	M 335.2	BOOL	// M-EINGANG: Schwenkfraeskopf Klemmung geklemmt
"I_SK_Klemmung_geloest"	M 335.3	BOOL	// M-EINGANG: Schwenkfraeskopf Klemmung geloest
"I_SPI_SCH_OELDRUCK_OK_1"	M 335.4	BOOL	// M-EINGANG: Druckueberwachung Schmierung Oel-Luftschmierung
"I_SPI_SCH_FUELLSTAND_OK"	M 335.5	BOOL	// M-EINGANG: Fuellstand Schmierstoffpumpe Oel-Luftschmierung
"I_SPI_SCH_LUFTDRUCK_OK"	M 335.6	BOOL	// M-EINGANG: Druckueberwachung Blasluft Getriebe Hauptantrieb
"I_SK_Freigabe"	M 335.7	BOOL	// M-EINGANG: Schwenkfräskopf Freigabe
"I_WM_Beladung_zu"	M 336.0	BOOL	// M-EINGANG: Fenster Werkzeugbestückung geschlossen
"I_WW_Uebergabeplatz"	M 336.1	BOOL	// M-EINGANG: Werkzeugmagazin Werkzeugerkennung Übergabeplatz
"I_WM_Zaehlimpuls"	M 336.2	BOOL	// M-EINGANG: Zaehlimpuls Werkzeugmagazin
"I_WM_Referenzimpuls"	M 336.3	BOOL	// M-EINGANG: Referenzimpuls Werkzeugmagazin
"I_WM_Energiefreigabe"	M 336.4	BOOL	// M-EINGANG: Werkzeugmagazin Energiefreigabe
"I_WA_ENABLE_LOCKED_CNC"	M 336.5	BOOL	// M-EINGANG: Taste Arbeitraum-Tuer verriegln
"I_WM_TAS_Beladung_auf"	M 336.6	BOOL	// M-EINGANG: Freigabe Magnetverriegelung WZB (Fenster Werkzeugbestückung) oeffnen
"I_WM_Taste_rechts"	M 336.7	BOOL	// M-EINGANG: Taste Kettenmagazin Plus-Richtung (rechts) fahren
"I_WM_Taste_links"	M 337.0	BOOL	// M-EINGANG: Taste Kettenmagazin Minus-Richtung (links) fahren
"I_PS_FRG_AR_PSACHS"	M 337.1	BOOL	// M-EINGANG: Antriebsfreigabe Arbeitsraum Palettenspeichersystem
"I_PS_NEG_NOT_AUS"	M 337.2	BOOL	// M-EINGANG: Rueckmeldung Not-Aus Palettenspeichersystem
"I_PS_BTB_PNOZ"	M 337.3	BOOL	// M-EINGANG: PNOZmulti Palettenspeichersystem betriebsbereit
"I_PS_FRG_AR_NCRPL"	M 337.4	BOOL	// M-EINGANG: Antriebsfreigabe Arbeitsraum Rüstplatz
"I_SF_NEG_UEBERLAUF"	M 337.5	BOOL	// M-EINGANG: Spaenefoerderer Ueberlaufbegrenzung Sammelbehaelter
"M_RS4_100_125er_Solution"	M 337.6	BOOL	// Merker Rundspeicher 4 für 100er/125er mit Solutionline
"I_WM_ZUSTIMMTASTE"	M 337.7	BOOL	// M-EINGANG: Zustimmtaste Magazin Zweihandbedienung
"I_WW_1_Klappe_zu"	M 338.0	BOOL	// M-EINGANG: Werkzeugwechsler Tuer geschlossen
"I_WW_Freigabe"	M 338.1	BOOL	// M-EINGANG: Freigabe Werkzeugwechsler
"I_AL_Druckluft_OK"	M 338.2	BOOL	// M-EINGANG: Druckueberwachung Druckluft (Systemdruck Pneumatik)
"I_WZ-Spanner_Gesp_O_WZ"	M 338.3	BOOL	// M-EINGANG: Werkzeugspanner gespannt ohne Werkzeug
"I_WZ_SPA_geloest"	M 338.4	BOOL	// M-EINGANG: Werkzeugspanner geloest
"I_WZ_SPA_gespannt"	M 338.5	BOOL	// M-EINGANG: Werkzeugspanner gespannt
"I_KM_NEG_MIN_FUELL"	M 338.6	BOOL	// M-EINGANG: Fuellstand Feinbereich Minimum
"I_KM_NEG_VOR_FUELL"	M 338.7	BOOL	// M-EINGANG: Kühlmittelanlage Kühlmittelmangel Feinbereich
"I_SF_UEBERLAUF"	M 339.0	BOOL	// M-EINGANG: Hebepumpe Spaenefoerderer Not-Aus
"I_WZB_Messung_Ende"	M 339.1	BOOL	// M-EINGANG: Werkzeugbruchüberwachung Messwertübernahme
"I_WZB_Bit_0"	M 339.2	BOOL	// M-EINGANG: Werkzeugbruchüberwachung BCD-Zahl 1
"I_WZB_Bit_1"	M 339.3	BOOL	// M-EINGANG: Werkzeugbruchüberwachung BCD-Zahl 2
"I_WZB_Bit_2"	M 339.4	BOOL	// M-EINGANG: Werkzeugbruchüberwachung BCD-Zahl 4
"I_WZB_Bit_3"	M 339.5	BOOL	// M-EINGANG: Werkzeugbruchüberwachung BCD-Zahl 8
"I_AL_3_Betriebsart"	M 339.6	BOOL	// M-EINGANG: Anwahl 3.Betriebsart
"I_AL_4_Betriebsart"	M 339.7	BOOL	// M-EINGANG: Anwahl 4.Betriebsart
"I_PW_Palette_geklemmt"	M 340.0	BOOL	// M-EINGANG: Palettenklemmung geklemmt
"I_PW_Klemmung_geloest"	M 340.1	BOOL	// M-EINGANG: Palettenklemmung geloest
"I_PW_Hub_unten"	M 340.2	BOOL	// M-EINGANG: Palettenwechsler Pos. unten
"I_PW_Ruestpl_Uebergabe"	M 340.3	BOOL	// M-EINGANG: Palettenwechsler Ruestplatz Wechselposition
"I_PW_Hub_oben"	M 340.4	BOOL	// M-EINGANG: Palettenwechsler Pos. oben
"I_PW_0_GRAD_M61"	M 340.5	BOOL	// M-EINGANG: 0 Grad Pos. Palettenwechsler
"I_PW_180_GRAD_M62"	M 340.6	BOOL	// M-EINGANG: 180 Grad Pos. Palettenwechsler
"I_PW_PAL_VORHANDEN"	M 340.7	BOOL	// M-EINGANG: Palettenwechsler Palette vorhanden
"I_PW_Tueren_zu"	M 341.0	BOOL	// M-EINGANG: Kabinentuer Drehpalettenwechsler geschlossen
"I_PW_ANDOCK_OBEN"	M 341.1	BOOL	// M-EINGANG: Palettenwechsler Rüstplatz Andockstation oben
"I_PW_PAL_GEKLEMMT"	M 341.2	BOOL	// M-EINGANG: Palettenwechsler Palette ist geklemmt
"I_Kab_Tuer_Entr"	M 341.3	BOOL	// M-EINGANG: Taste Kabinentür entriegeln
"I_PW_AUF_RP_GESPANNT"	M 341.4	BOOL	// M-EINGANG: Palettenwechsler Palette auf  Ruestplatz gespannt
"I_MSST_WM_Taste_Rechts"	M 341.5	BOOL	// M-EINGANG: Taste Werkzeugmagazin rechts
"I_MSST_WM_Taste_links"	M 341.6	BOOL	// M-EINGANG: Taste Werkzeugmagazin links
"I_PW_AUF_RP_GELOEST"	M 341.7	BOOL	// M-EINGANG: Palette auf Rüstplatz gelöst
"I_HR_Achsanwahl_Bit_0"	M 342.0	BOOL	// M-EINGANG: GRAY-Code Achsumschaltung Bit 0
"I_HR_Achsanwahl_Bit_1"	M 342.1	BOOL	// M-EINGANG: GRAY-Code Achsumschaltung Bit 1
"I_HR_Achsanwahl_Bit_2"	M 342.2	BOOL	// M-EINGANG: GRAY-Code Achsumschaltung Bit 2
"I_HR_plus_Taste"	M 342.3	BOOL	// M-EINGANG: Handrad Taste +
"I_HR_minus_Taste"	M 342.4	BOOL	// M-EINGANG: Handrad Taste -
"I_HR_Eilgang_Taste"	M 342.5	BOOL	// M-EINGANG: Handrad Taste Eilgang
"I_HR_FKT_Taste_F1"	M 342.6	BOOL	// M-EINGANG: Handrad Taste F1
"I_HR_FKT_Taste_F2"	M 342.7	BOOL	// M-EINGANG: Handrad Taste F2
"I_HR_FKT_Taste_F3"	M 343.0	BOOL	// M-EINGANG: Handrad Taste F3
"I_WW_Rueck_hlt_AUSGEF"	M 343.1	BOOL	// M-EINGANG: Werkzeug-Rueckhalt ausgefahren (verriegeln)
"I_WW_Rueck_hlt_GST"	M 343.2	BOOL	// M-EINGANG: Werkzeug-Rueckhalt in Grundstellung
"I_WW_Rein_in_Rein_Pos"	M 343.3	BOOL	// M-EINGANG: Reinigung Werkzeugkegel ausgefahren
"I_WW_Rein_in_GST"	M 343.4	BOOL	// M-EINGANG: Reinigung Werkzeugkegel eingefahren
"I_LA_ausgefahren"	M 343.5	BOOL	// M-EINGANG: LA: Laser ausgefahren
"I_LA_eingeschwenkt"	M 343.6	BOOL	// M-EINGANG: LA: Laser eingefahren
"I_LA_BTB"	M 343.7	BOOL	// M-EINGANG: LA: Laser ok
"I_LA_statisches_Signal"	M 344.0	BOOL	// M-EINGANG: LA: Laser Signal statisch
"I_LA_Klappe_zu"	M 344.1	BOOL	// M-EINGANG: Laser: Schmutzblende geschlossen
"I_AL_NEG_Not_Aus"	M 344.2	BOOL	// M-EINGANG: Rueckmeldung Maschine Ein (Kein Not-Aus)
"I_AL_ACHS_Drehzahl_OK"	M 344.3	BOOL	// M-EINGANG: Ueberwachung Drehzahlbegrenzung
"M_Read_AccessLevel"	M 344.4	BOOL	// Start des Lesevorgangs zur Ermittlung des AccessLevel aus den NC-Daten
"M_RADMAGAZIN"	M 344.5	BOOL	// Radmagazin
"M_Req_write_Bruchdaten"	M 344.6	BOOL	// Anforderung Bruchdaten schreiben
"O_AL_NEG_POWERSAVE_STBY"	M 344.7	BOOL	// M-AUSGANG: Maschinenabschaltung
"M_KSS_TEMP_ZU_HOCH"	M 345.0	BOOL	// KM: Kühlschmierstoff Temperatur zu hoch
"MX_WZ_BRUCH_LASER"	M 345.1	BOOL	// Werkzeugbruch erkannt durch Laser
"M_VERTIKALKETTE"	M 345.2	BOOL	// Vertikalkette
"M_TagRemoved"	M 345.3	BOOL	// Angelegter Smartkey wurde entfernt
"M_NewTagInside"	M 345.4	BOOL	// Neuer Smartkey wurde angelegt und erkannt
"M_FP_TagRemoved"	M 345.5	BOOL	// Positive Flanke von Smartkey wurde entfernt
"M_Freigab_ZD_WZW"	M 345.6	BOOL	// SAFETY: Freigabe an WZW
"M_Anf_ZD_WZW"	M 345.7	BOOL	// SAFETY: Anforderung Zwangsdynamisisierung von  WZW steht an
"I_Taste_ToFrame"	M 346.0	BOOL	// M-EINGANG: MSST-Taste ToFrame
"I_4Ax_Klemm_Auf"	M 346.1	BOOL	// M-EINGANG: Klemmung 4. Achse gelöst
"I_5Ax_Klemm_Auf"	M 346.2	BOOL	// M-EINGANG: Klemmung 5. Achse gelöst
"I_AL_Sternschaltung"	M 346.3	BOOL	// M-EINGANG: Eingang Sternschaltung
"I_AL_Dreieckschaltung"	M 346.4	BOOL	// M-EINGANG: Eingang Dreieckschaltung
"MX_T_WZ_DREHMOMENT_STOP"	M 346.5	BOOL	// WZV: Drehmomentueberwachung Tol 2 hat angesprochen (Fehler 67111)
"MX_T_WZ_Drehmoment"	M 346.6	BOOL	// WZV: Drehmomentueberwachung Tol 1 hat angesprochen (Fehler 65109)
"MX_T_WZ_Standzeit"	M 346.7	BOOL	// WZV: Werkzeugstandzeit abgelaufen
"I_KA_NEG_Sammelfehler"	M 347.0	BOOL	// M-EINGANG: Kuehlaggregat Stoerung
"I_Fehler_KA_Fuellst"	M 347.1	BOOL	// M-EINGANG: Störmeldung Kühlaggregat Füllstand
"I_KA_NEG_Luftfilter"	M 347.2	BOOL	// M-EINGANG: Kühlaggregat Störmeldung Filterverschmutzung
"I_PW_RP_TUER_1_OFFEN"	M 347.3	BOOL	// M-EINGANG: Rüstplatz-Tür 1 (links) offen
"I_PW_RP_TUER_2_OFFEN"	M 347.4	BOOL	// M-EINGANG: Rüstplatz-Tür 2 (rechts) offen
"I_RPL_T_DREHEN"	M 347.5	BOOL	// M-EINGANG: Taste Rüstplatz-Achse drehen
"I_RPL_T_ZUSTIMM"	M 347.6	BOOL	// M-EINGANG: Zustimm-Taste am Rüstplatz
"O_RPL_TUER_OEFFNEN"	M 347.7	BOOL	// M-AUSGANG: Ventil Rüstplatztür öffnen
"I_PS_RPL_TUER_VORN_VERR"	M 352.0	BOOL	// M-EINGANG: Ruestplatztuer Palettenspeichersystem verriegelt vorn
"I_PS_RPL_TUER_HINT_VERR"	M 352.1	BOOL	// M-EINGANG: Ruestplatztuer Palettenspeichersystem verriegelt hinten
"I_PS_RPL_TUER_VORNE_ZU"	M 352.2	BOOL	// M-EINGANG: Ruestplatztuer vorn geschlossen
"I_PS_RPL_TUER_HINTEN_ZU"	M 352.3	BOOL	// M-EINGANG: Ruestplatztuer hinten geschlossen
"I_D_PS_RPL_PAL_VORH"	M 352.4	BOOL	// M-EINGANG: Palette Ruestplatz vorhanden Diagnose
"I_PS_RPL_PAL_VORH"	M 352.5	BOOL	// M-EINGANG: Palette Ruestplatz vorhanden
"I_PS_RPL_GST"	M 352.6	BOOL	// M-EINGANG: Ruestplatz Palettenspeichersystem Grundstellung
"I_AL_Hubtuere_zu"	M 352.7	BOOL	// M-EINGANG: Hubtuere Palettenwechsel Sicherheitsschalter
"I_PS_DREHST_PAL_GST"	M 353.0	BOOL	// M-EINGANG: Palette auf Schlitten vorhanden Drehachse
"I_PS_DREHST_PAL_VORH"	M 353.1	BOOL	// M-EINGANG: Ueberwachung Palette vorhanden Ablageplatz
"I_D_PS_DREHST_PAL_VORH"	M 353.2	BOOL	// M-EINGANG: Ueberwachung Palette vorhanden Ablageplatz Öffner
"I_PS_DREHBER_OK"	M 353.3	BOOL	// M-EINGANG: Meldung Drehbereichsbegrenzung betaetigt
"I_PS_DREHST_HUB_UNTEN"	M 353.4	BOOL	// M-EINGANG: Sensor Dreheinheit unten
"I_PS_DREHST_HUB_OBEN"	M 353.5	BOOL	// M-EINGANG: Sensor Dreheinheit oben
"I_PW_RPL_Gespannt"	M 353.6	BOOL	// M-EINGANG:
"I_RP_Rohteil_setzen"	M 353.7	BOOL	// M-EINGANG:
"M_WZM_Regal_angewaehlt"	M 354.0	BOOL	// WZW: OMRON-Regalmagazin angewaehlt
"I_AL_AR3_OK"	M 354.1	BOOL	// M-EINGANG:
"I_SP_AUFL_ST1_GESPANNT"	M 354.2	BOOL	// M-EINGANG: Kontrolle Auflage Spannstelle 1 gespannt ok
"I_SP_AUFL_ST2_GESPANNT"	M 354.3	BOOL	// M-EINGANG: Kontrolle Auflage Spannstelle 2 gespannt ok
"I_SP_AUFL_ST3_GESPANNT"	M 354.4	BOOL	// M-EINGANG: Kontrolle Auflage Spannstelle 3 gespannt ok
"I_SP_AUFL_ST4_GESPANNT"	M 354.5	BOOL	// M-EINGANG: Kontrolle Auflage Spannstelle 4 gespannt ok
"I_SP_HYD_FUELL_MIN_OK"	M 354.6	BOOL	// M-EINGANG: Spannhydraulik Fuellstand ok
"I_SP_MPL_ENTKUPPELT"	M 354.7	BOOL	// M-EINGANG: Spannhydraulik Maschinenplatz entkuppelt
"I_PW_MPL_MDK_ENTKUPPELT"	M 355.0	BOOL	// M-EINGANG: Medienkupplung Fraes-Drehtisch eingefahren
"I_SP_MPL_GEKUPPELT"	M 355.1	BOOL	// M-EINGANG: Spannhydraulik Maschinenplatz gekuppelt
"I_SP_RPL_ENTKUPPELT"	M 355.2	BOOL	// M-EINGANG: Spannhydraulik Rüstplatz entkuppelt
"I_SP_RPL_GEKUPPELT"	M 355.3	BOOL	// M-EINGANG: Spannhydraulik Rüstplatz gekuppelt
"I_SP_T_SPANNSTELLE_1"	M 355.4	BOOL	// M-EINGANG: Spannhydraulik Taster Spannstelle 1
"I_SP_T_SPANNSTELLE_2"	M 355.5	BOOL	// M-EINGANG: Spannhydraulik Taster Spannstelle 2
